C07129=5344,30396,-30623,463,-27004,-2829
C07130=5352,30386,-30635,462,-27000,-2833
C07131=5354,30373,-30650,461,-26996,-2833
C07132=5355,30360,-30666,461,-26991,-2834
C07133=5361,30350,-30679,461,-26987,-2836
C07134=5368,30340,-30691,460,-26983,-2839
C07135=5370,30327,-30707,459,-26978,-2840
C07136=5374,30315,-30721,459,-26974,-2841
C07137=5383,30306,-30731,458,-26971,-2845
C07138=5385,30293,-30747,457,-26966,-2846
C07139=5393,30284,-30758,456,-26963,-2849
C07140=5398,30273,-30772,456,-26958,-2851
C07141=5409,30265,-30781,454,-26956,-2855
C07142=5413,30254,-30795,454,-26951,-2857
C07143=5422,30245,-30806,452,-26948,-2860
C07144=5428,30234,-30818,451,-26944,-2863
C07145=5428,30229,-30825,451,-26942,-2863
C07146=5414,30227,-30827,454,-26941,-2857
C07147=5410,30239,-30813,454,-26946,-2856
C07148=5399,30246,-30804,456,-26949,-2851
C07149=5389,30255,-30793,457,-26952,-2848
C07150=5388,30268,-30778,457,-26957,-2847
C07151=5379,30277,-30767,458,-26960,-2843
C07152=5379,30277,-29367,458,-26960,-2843
C07153=5291,30621,-26350,469,-27087,-2808
C07154=5291,30621,-30350,469,-27087,-2808
C07155=5290,30633,-30335,469,-27092,-2807
C07156=5284,30643,-30323,470,-27096,-2805
C07157=5277,30652,-30312,471,-27099,-2802
C07158=5275,30665,-30298,471,-27104,-2802
C07159=5266,30673,-30288,472,-27107,-2798
C07160=5263,30684,-30275,473,-27111,-2797
C07161=5259,30695,-30261,473,-27115,-2795
C07162=5250,30703,-30251,474,-27118,-2792
C07163=5245,30713,-30239,475,-27121,-2790
C07164=5237,30722,-30228,476,-27125,-2787
C07165=5236,30734,-30214,476,-27129,-2786
C07166=5234,30746,-30199,476,-27134,-2785
C07167=5224,30754,-30190,478,-27136,-2781
C07168=5221,30765,-30176,478,-27141,-2780
C07169=5217,30776,-30163,479,-27145,-2778
C07170=5209,30785,-30153,480,-27148,-2775
C07171=5207,30797,-30138,480,-27152,-2775
C07172=5206,30809,-30123,480,-27157,-2774
C07173=5196,30817,-30114,482,-27160,-2770
C07174=5193,30828,-28700,482,-27164,-2769
C07175=-41004,59868,4099,4900,-34257,16705
C07176=-41004,59868,1099,4900,-34257,16705
C07177=-41004,64596,1380,5213,-31659,16463
C07178=-41004,59868,1099,4900,-34257,16705
C07179=-41004,59868,9099,4900,-34257,16705
C07180=5193,30828,-26100,482,-27164,-2769
C07181=5193,30828,-30100,482,-27164,-2769
C07182=5191,30840,-30085,482,-27168,-2768
C07183=5190,30853,-30070,482,-27173,-2768
C07184=5188,30865,-30055,482,-27178,-2767
C07185=5178,30872,-30047,484,-27180,-2763
C07186=5175,30884,-30032,484,-27185,-2762
C07187=5174,30896,-30018,484,-27189,-2761
C07188=5172,30908,-30003,484,-27194,-2761
C07189=5171,30921,-29988,484,-27198,-2760
C07190=5169,30933,-29973,485,-27203,-2759
C07191=5174,30934,-29971,484,-27203,-2761
C07192=5181,30925,-29983,483,-27200,-2764
C07193=5182,30913,-29997,483,-27195,-2764
C07194=5184,30900,-30012,483,-27191,-2765
C07195=5185,30888,-30027,483,-27186,-2766
C07196=5192,30879,-30038,482,-27183,-2768
C07197=5198,30869,-30050,481,-27179,-2771
C07198=5200,30857,-30065,481,-27175,-2771
C07199=5201,30845,-30080,481,-27170,-2772
C07200=5207,30835,-30092,480,-27166,-2774
C07201=5214,30826,-30103,479,-27163,-2777
C07202=5215,30813,-30118,479,-27159,-2778
C07203=5217,30801,-30132,478,-27154,-2779
C07204=5228,30794,-30141,477,-27151,-2783
C07205=5230,30782,-30156,477,-27147,-2783
C07206=5235,30772,-30168,476,-27143,-2785
C07207=5242,30763,-30179,475,-27140,-2788
C07208=5244,30751,-30193,475,-27135,-2789
C07209=5253,30742,-30203,474,-27132,-2792
C07210=5257,30732,-30217,473,-27128,-2794
C07211=5260,30720,-30230,473,-27124,-2795
C07212=5269,30712,-30240,471,-27121,-2799
C07213=5271,30700,-30254,471,-27117,-2800
C07214=5277,30691,-30266,470,-27113,-2802
C07215=5284,30681,-30278,470,-27110,-2805
C07216=5285,30669,-30292,469,-27105,-2805
C07217=5288,30657,-30306,469,-27101,-2807
C07218=5298,30650,-30315,468,-27098,-2810
C07219=5300,30638,-30330,468,-27094,-2811
C07220=5301,30625,-30345,467,-27089,-2812
C07221=5291,30621,-30350,469,-27087,-2808
C07222=5291,30621,-28950,469,-27087,-2808
C07223=5528,30636,-26331,434,-27095,-2900
C07224=5528,30636,-30331,434,-27095,-2900
C07225=5527,30651,-30313,434,-27101,-2899
C07226=5525,30666,-30295,434,-27106,-2898
C07227=5523,30681,-30277,435,-27112,-2897
C07228=5512,30691,-30265,436,-27115,-2893
C07229=5509,30705,-30248,436,-27121,-2892
C07230=5500,30716,-30234,438,-27124,-2888
C07231=5496,30729,-30218,438,-27129,-2887
C07232=5494,30744,-30200,438,-27135,-2886
C07233=5483,30754,-30189,440,-27138,-2881
C07234=5477,30766,-30173,441,-27143,-2879
C07235=5469,30778,-30160,442,-27147,-2876
C07236=5465,30792,-30143,442,-27152,-2875
C07237=5455,30802,-30130,444,-27156,-2871
C07238=5453,30817,-30112,444,-27162,-2870
C07239=5442,30826,-30101,445,-27165,-2865
C07240=5440,30841,-30083,446,-27171,-2865
C07241=5429,30851,-30071,447,-27174,-2860
C07242=5426,30865,-30054,447,-27180,-2859
C07243=5417,30876,-30041,449,-27184,-2856
C07244=5412,30889,-30025,449,-27188,-2853
C07245=5401,30899,-30013,451,-27192,-2849
C07246=5399,30914,-29995,451,-27198,-2849
C07247=5394,30927,-29979,452,-27202,-2846
C07248=5386,30938,-29966,453,-27206,-2843
C07249=5384,30953,-29948,453,-27212,-2842
C07250=5382,30968,-29930,453,-27218,-2842
C07251=5391,30980,-29915,452,-27222,-2845
C07252=5389,30995,-29897,452,-27228,-2844
C07253=5387,31010,-29879,452,-27233,-2843
C07254=5392,31014,-29874,452,-27235,-2845
C07255=5399,31002,-29888,451,-27230,-2848
C07256=5400,30987,-29906,450,-27225,-2849
C07257=5402,30972,-29924,450,-27219,-2849
C07258=5404,30957,-29942,450,-27214,-2850
C07259=5406,30942,-29960,450,-27208,-2851
C07260=5413,30930,-29975,449,-27204,-2854
C07261=5420,30918,-29990,448,-27199,-2856
C07262=5421,30903,-30007,448,-27194,-2857
C07263=5431,30893,-30020,447,-27190,-2861
C07264=5435,30879,-30037,446,-27185,-2862
C07265=5442,30867,-30051,445,-27181,-2865
C07266=5448,30855,-30066,444,-27176,-2868
C07267=5454,30842,-30082,444,-27171,-2870
C07268=5462,30831,-30095,443,-27167,-2873
C07269=5466,30817,-30112,442,-27162,-2875
C07270=5475,30806,-30125,441,-27158,-2878
C07271=5484,30795,-30138,439,-27154,-2882
C07272=5489,30782,-30154,439,-27149,-2884
C07273=5496,30770,-30169,438,-27145,-2887
C07274=5502,30758,-30183,437,-27140,-2889
C07275=5508,30745,-30199,436,-27135,-2891
C07276=5516,30734,-30213,435,-27131,-2894
C07277=5519,30720,-30230,435,-27126,-2896
C07278=5529,30709,-30242,433,-27122,-2900
C07279=5531,30695,-30260,433,-27117,-2901
C07280=5537,30682,-30276,433,-27112,-2903
C07281=5545,30670,-30289,431,-27108,-2906
C07282=5547,30656,-30307,431,-27102,-2907
C07283=5542,30642,-30324,432,-27097,-2905
C07284=5528,30636,-30331,434,-27095,-2900
C07285=5528,30636,-28931,434,-27095,-2900
C07286=5871,30873,-26043,382,-27186,-3031
C07287=5871,30873,-30043,382,-27186,-3031
C07288=5877,30878,-30036,381,-27188,-3034
C07289=5889,30880,-30034,380,-27189,-3038
C07290=5901,30882,-30031,378,-27190,-3043
C07291=5912,30883,-30029,376,-27190,-3047
C07292=5924,30885,-30027,375,-27191,-3052
C07293=5936,30887,-30025,373,-27192,-3056
C07294=5947,30888,-30023,371,-27193,-3061
C07295=5959,30890,-30021,369,-27193,-3065
C07296=5971,30892,-30019,368,-27194,-3070
C07297=5982,30894,-30017,366,-27195,-3074
C07298=5994,30895,-30015,364,-27195,-3079
C07299=6006,30897,-30012,363,-27196,-3083
C07300=6018,30899,-30010,361,-27197,-3088
C07301=6029,30900,-30008,359,-27198,-3093
C07302=6041,30902,-30006,357,-27198,-3097
C07303=6053,30904,-30004,356,-27199,-3102
C07304=6064,30906,-30002,354,-27200,-3106
C07305=6071,30914,-29991,353,-27203,-3109
C07306=6079,30923,-29980,352,-27207,-3112
C07307=6081,30933,-29968,351,-27210,-3112
C07308=6080,30944,-29955,351,-27214,-3112
C07309=6078,30955,-29942,352,-27218,-3111
C07310=6069,30961,-29934,353,-27221,-3108
C07311=6060,30968,-29926,354,-27223,-3104
C07312=6054,30976,-29916,355,-27226,-3102
C07313=6053,30987,-29903,355,-27230,-3101
C07314=6051,30998,-29890,355,-27234,-3101
C07315=6061,31001,-29886,354,-27235,-3105
C07316=6071,30994,-29894,352,-27233,-3108
C07317=6080,30988,-29902,351,-27231,-3112
C07318=6089,30981,-29910,350,-27228,-3116
C07319=6099,30975,-29917,348,-27226,-3119
C07320=6107,30968,-29925,347,-27224,-3122
C07321=6099,30960,-29936,348,-27220,-3119
C07322=6100,30949,-29949,349,-27216,-3120
C07323=6101,30938,-29962,348,-27212,-3120
C07324=6100,30928,-29974,349,-27209,-3120
C07325=6093,30919,-29985,350,-27205,-3117
C07326=6095,30908,-29998,349,-27201,-3118
C07327=6093,30900,-30008,350,-27198,-3117
C07328=6081,30898,-30011,352,-27197,-3113
C07329=6072,30893,-30017,353,-27195,-3109
C07330=6063,30886,-30025,354,-27193,-3106
C07331=6051,30884,-30027,356,-27192,-3101
C07332=6040,30883,-30030,358,-27191,-3097
C07333=6028,30881,-30032,359,-27190,-3092
C07334=6016,30879,-30034,361,-27190,-3088
C07335=6005,30878,-30036,363,-27189,-3083
C07336=5993,30876,-30038,365,-27188,-3079
C07337=5981,30874,-30040,366,-27188,-3074
C07338=5969,30873,-30042,368,-27187,-3069
C07339=5958,30871,-30044,370,-27186,-3065
C07340=5946,30869,-30046,371,-27185,-3060
C07341=5934,30867,-30049,373,-27185,-3056
C07342=5925,30874,-30041,374,-27187,-3052
C07343=5914,30874,-30041,376,-27187,-3048
C07344=5902,30872,-30043,378,-27186,-3043
C07345=5890,30871,-30045,380,-27185,-3039
C07346=5879,30869,-30047,381,-27185,-3034
C07347=5871,30873,-28643,382,-27186,-3031
C07348=-41004,59868,4099,4900,-34257,16705
C07349=-41004,59868,1099,4900,-34257,16705
C07350=-41004,64596,1380,5213,-31659,16463
C07351=-41004,59868,1099,4900,-34257,16705
C07352=-41004,59868,9099,4900,-34257,16705
C07353=5871,30873,-26043,382,-27186,-3031
C07354=5871,30873,-30043,382,-27186,-3031
C07355=5871,30873,-28643,382,-27186,-3031
C07356=5732,31221,-25621,401,-27315,-2976
C07357=5732,31221,-29621,401,-27315,-2976
C07358=5695,31216,-29627,406,-27313,-2962
C07359=5657,31210,-29634,412,-27310,-2947
C07360=5620,31205,-29641,417,-27308,-2933
C07361=5583,31200,-29648,422,-27306,-2918
C07362=5546,31194,-29654,428,-27303,-2904
C07363=5509,31189,-29661,433,-27301,-2890
C07364=5475,31193,-29656,438,-27303,-2876
C07365=5437,31188,-29662,444,-27300,-2862
C07366=5401,31187,-29664,449,-27300,-2848
C07367=5366,31187,-29664,454,-27299,-2834
C07368=5332,31193,-29657,459,-27301,-2821
C07369=5298,31196,-29653,464,-27302,-2808
C07370=5264,31201,-29647,469,-27304,-2795
C07371=5229,31206,-29642,474,-27305,-2781
C07372=5196,31211,-29635,479,-27307,-2768
C07373=5164,31225,-29619,483,-27312,-2756
C07374=5130,31230,-29614,488,-27313,-2743
C07375=5099,31244,-29596,493,-27318,-2731
C07376=5065,31249,-29591,498,-27320,-2717
C07377=5032,31258,-29580,502,-27323,-2705
C07378=5000,31268,-29568,507,-27326,-2692
C07379=4967,31278,-29556,512,-27330,-2679
C07380=4945,31289,-29543,515,-27334,-2671
C07381=4979,31284,-29548,510,-27332,-2684
C07382=5011,31272,-29562,505,-27328,-2696
C07383=5045,31265,-29571,500,-27326,-2709
C07384=5079,31260,-29577,496,-27324,-2723
C07385=5112,31253,-29585,491,-27322,-2736
C07386=5144,31241,-29600,486,-27318,-2748
C07387=5178,31236,-29605,481,-27316,-2761
C07388=5212,31232,-29610,476,-27315,-2774
C07389=5246,31227,-29616,471,-27313,-2788
C07390=5280,31223,-29621,466,-27312,-2801
C07391=5314,31218,-29627,461,-27310,-2814
C07392=5349,31213,-29632,457,-27309,-2827
C07393=5385,31216,-29629,451,-27310,-2842
C07394=5420,31214,-29631,446,-27310,-2855
C07395=5454,31210,-29636,441,-27309,-2868
C07396=5490,31211,-29635,436,-27309,-2882
C07397=5525,31210,-29635,431,-27309,-2896
C07398=5563,31216,-29628,425,-27312,-2910
C07399=5600,31221,-29621,420,-27314,-2925
C07400=5637,31227,-29615,414,-27316,-2939
C07401=5674,31232,-29608,409,-27319,-2954
C07402=5711,31237,-29601,404,-27321,-2968
C07403=5748,31243,-29594,398,-27323,-2982
C07404=5785,31248,-29588,393,-27326,-2997
C07405=5823,31254,-29581,387,-27328,-3011
C07406=5854,31268,-29564,382,-27334,-3023
C07407=5892,31273,-29557,377,-27336,-3038
C07408=5923,31287,-29539,372,-27341,-3050
C07409=5960,31293,-29532,367,-27344,-3064
C07410=5974,31288,-29538,365,-27342,-3070
C07411=5939,31279,-29550,370,-27338,-3056
C07412=5907,31266,-29566,375,-27333,-3044
C07413=5875,31252,-29583,380,-27328,-3031
C07414=5838,31246,-29590,385,-27325,-3017
C07415=5801,31240,-29597,390,-27323,-3003
C07416=5769,31227,-29614,395,-27317,-2990
C07417=5732,31221,-29621,401,-27315,-2976
C07418=5732,31221,-28221,401,-27315,-2976
C07419=4765,31119,-25749,542,-27269,-2602
C07420=4765,31119,-29749,542,-27269,-2602
C07421=4766,31110,-29761,542,-27265,-2602
C07422=4760,31102,-29770,543,-27262,-2600
C07423=4758,31094,-29780,543,-27259,-2599
C07424=4759,31085,-29791,543,-27256,-2599
C07425=4760,31075,-29802,543,-27252,-2600
C07426=4764,31068,-29811,543,-27250,-2602
C07427=4772,31062,-29818,542,-27248,-2605
C07428=4773,31053,-29829,542,-27244,-2605
C07429=4763,31052,-29831,543,-27244,-2601
C07430=4755,31057,-29824,544,-27246,-2598
C07431=4751,31065,-29815,545,-27248,-2596
C07432=4750,31074,-29804,545,-27252,-2596
C07433=4749,31083,-29793,545,-27255,-2595
C07434=4747,31093,-29782,545,-27259,-2595
C07435=4746,31102,-29770,545,-27262,-2595
C07436=4745,31111,-29759,545,-27266,-2594
C07437=4744,31120,-29748,545,-27269,-2594
C07438=4743,31129,-29737,545,-27272,-2593
C07439=4739,31137,-29728,546,-27275,-2592
C07440=4732,31143,-29721,547,-27277,-2589
C07441=4730,31152,-29710,547,-27281,-2588
C07442=4729,31161,-29699,547,-27284,-2588
C07443=4722,31167,-29692,548,-27286,-2585
C07444=4717,31174,-29683,549,-27289,-2583
C07445=4713,31182,-29674,549,-27292,-2581
C07446=4705,31187,-29667,550,-27294,-2578
C07447=4704,31196,-29656,550,-27297,-2578
C07448=4697,31202,-29649,551,-27299,-2575
C07449=4693,31210,-29640,552,-27302,-2573
C07450=4688,31217,-29631,553,-27305,-2571
C07451=4681,31223,-29624,554,-27307,-2568
C07452=4679,31232,-29614,554,-27310,-2568
C07453=4671,31237,-29607,555,-27312,-2565
C07454=4668,31245,-29597,555,-27315,-2563
C07455=4663,31252,-29589,556,-27317,-2561
C07456=4656,31258,-29582,557,-27320,-2559
C07457=4655,31267,-29570,557,-27323,-2558
C07458=4655,31274,-29562,557,-27326,-2558
C07459=4663,31269,-29568,556,-27324,-2561
C07460=4671,31263,-29575,555,-27322,-2564
C07461=4677,31257,-29583,554,-27319,-2567
C07462=4679,31249,-29593,554,-27316,-2568
C07463=4687,31243,-29600,553,-27314,-2571
C07464=4690,31235,-29610,552,-27311,-2572
C07465=4696,31228,-29617,551,-27309,-2574
C07466=4701,31222,-29626,551,-27306,-2576
C07467=4705,31214,-29635,550,-27303,-2578
C07468=4712,31208,-29642,549,-27301,-2581
C07469=4714,31199,-29653,549,-27298,-2582
C07470=4721,31193,-29660,548,-27296,-2584
C07471=4726,31186,-29668,547,-27293,-2586
C07472=4730,31178,-29678,547,-27291,-2588
C07473=4738,31173,-29684,546,-27289,-2591
C07474=4739,31164,-29695,546,-27285,-2591
C07475=4746,31158,-29702,545,-27283,-2594
C07476=4751,31151,-29711,544,-27280,-2596
C07477=4752,31141,-29722,544,-27277,-2597
C07478=4753,31132,-29734,544,-27274,-2597
C07479=4757,31125,-29743,543,-27271,-2599
C07480=4765,31119,-29749,542,-27269,-2602
C07481=4765,31119,-28349,542,-27269,-2602
C07482=3339,30279,-26773,757,-26945,-2054
C07483=3339,30279,-30773,757,-26945,-2054
C07484=3349,30265,-30790,756,-26939,-2058
C07485=3361,30252,-30806,754,-26935,-2062
C07486=3371,30239,-30822,753,-26930,-2067
C07487=3380,30224,-30840,752,-26924,-2070
C07488=3386,30208,-30860,751,-26918,-2072
C07489=3397,30194,-30876,750,-26914,-2077
C07490=3405,30180,-30894,749,-26908,-2080
C07491=3413,30165,-30911,748,-26903,-2083
C07492=3416,30152,-30927,747,-26898,-2084
C07493=3411,30135,-30947,748,-26892,-2082
C07494=3405,30119,-30968,749,-26885,-2080
C07495=3396,30103,-30987,751,-26879,-2077
C07496=3387,30087,-31006,752,-26873,-2074
C07497=3389,30068,-31028,752,-26867,-2075
C07498=3391,30050,-31051,752,-26860,-2075
C07499=3393,30031,-31073,752,-26853,-2076
C07500=3394,30013,-31095,752,-26846,-2077
C07501=3402,29998,-31114,751,-26841,-2080
C07502=3408,29982,-31133,750,-26835,-2082
C07503=3410,29963,-31155,750,-26828,-2083
C07504=3411,29945,-31178,750,-26821,-2084
C07505=3413,29926,-31200,750,-26814,-2085
C07506=3415,29908,-31222,750,-26807,-2086
C07507=3424,29894,-31239,749,-26802,-2089
C07508=3429,29877,-31260,748,-26796,-2091
C07509=3430,29858,-31282,748,-26789,-2092
C07510=3432,29840,-31304,748,-26782,-2093
C07511=3430,29822,-31326,748,-26776,-2092
C07512=3414,29813,-31336,751,-26772,-2086
C07513=3412,29832,-31314,751,-26779,-2085
C07514=3410,29850,-31292,751,-26786,-2084
C07515=3408,29869,-31270,751,-26793,-2083
C07516=3407,29887,-31248,751,-26800,-2083
C07517=3405,29905,-31225,751,-26806,-2082
C07518=3398,29921,-31206,752,-26812,-2079
C07519=3391,29937,-31187,753,-26818,-2076
C07520=3390,29955,-31165,753,-26825,-2076
C07521=3388,29974,-31143,753,-26832,-2075
C07522=3385,29992,-31121,753,-26838,-2074
C07523=3374,30005,-29705,755,-26843,-2069
C07524=-41004,59868,4099,4900,-34257,16705
C07525=-41004,59868,1099,4900,-34257,16705
C07526=-41004,64596,1380,5213,-31659,16463
C07527=-41004,59868,1099,4900,-34257,16705
C07528=-41004,59868,9099,4900,-34257,16705
C07529=3374,30005,-27105,755,-26843,-2069
C07530=3374,30005,-31105,755,-26843,-2069
C07531=3373,30023,-31083,755,-26850,-2069
C07532=3371,30042,-31060,755,-26857,-2068
C07533=3369,30060,-31038,755,-26864,-2067
C07534=3367,30079,-31016,755,-26870,-2066
C07535=3366,30097,-30994,755,-26877,-2065
C07536=3374,30113,-30974,754,-26883,-2068
C07537=3387,30128,-30956,752,-26889,-2073
C07538=3392,30145,-30936,751,-26895,-2075
C07539=3397,30159,-30919,750,-26900,-2077
C07540=3389,30174,-30901,751,-26906,-2074
C07541=3378,30187,-30885,753,-26911,-2069
C07542=3372,30203,-30865,753,-26917,-2067
C07543=3364,30218,-30847,754,-26922,-2064
C07544=3355,30233,-30830,755,-26927,-2060
C07545=3341,30244,-30816,757,-26932,-2055
C07546=3331,30258,-30799,759,-26937,-2051
C07547=3327,30276,-30778,759,-26943,-2049
C07548=3316,30289,-30762,761,-26948,-2045
C07549=3324,30290,-30760,759,-26948,-2048
C07550=3339,30279,-30773,757,-26945,-2054
C07551=3339,30279,-29373,757,-26945,-2054
C07552=3255,30276,-26778,770,-26943,-2021
C07553=3255,30276,-30778,770,-26943,-2021
C07554=3257,30254,-30805,770,-26934,-2022
C07555=3266,30235,-30827,768,-26928,-2026
C07556=3271,30215,-30852,768,-26920,-2028
C07557=3282,30197,-30873,766,-26914,-2032
C07558=3283,30177,-30897,766,-26906,-2033
C07559=3263,30185,-30888,769,-26909,-2025
C07560=3246,30184,-30889,772,-26908,-2018
C07561=3245,30162,-30916,772,-26900,-2018
C07562=3247,30140,-30942,772,-26892,-2019
C07563=3249,30118,-30969,772,-26884,-2020
C07564=3259,30099,-30991,771,-26877,-2024
C07565=3273,30084,-31010,769,-26872,-2030
C07566=3275,30062,-31037,769,-26863,-2031
C07567=3267,30042,-31061,770,-26856,-2028
C07568=3260,30022,-31085,771,-26848,-2025
C07569=3261,30000,-31112,772,-26840,-2025
C07570=3263,29978,-31138,771,-26832,-2026
C07571=3265,29956,-31165,771,-26824,-2027
C07572=3276,29938,-31186,770,-26818,-2032
C07573=3279,29917,-31212,770,-26810,-2033
C07574=3281,29894,-31239,770,-26801,-2034
C07575=3273,29875,-31263,771,-26794,-2031
C07576=3275,29852,-31290,771,-26786,-2032
C07577=3268,29832,-31314,772,-26778,-2029
C07578=3260,29812,-31339,774,-26771,-2026
C07579=3259,29791,-31365,774,-26763,-2026
C07580=3240,29779,-31379,777,-26758,-2019
C07581=3241,29800,-31353,776,-26766,-2019
C07582=3249,29820,-31329,775,-26774,-2022
C07583=3255,29841,-31304,774,-26781,-2024
C07584=3253,29863,-31278,774,-26789,-2023
C07585=3251,29885,-31251,774,-26798,-2022
C07586=3249,29907,-31224,774,-26806,-2021
C07587=3246,29929,-31197,774,-26814,-2020
C07588=3244,29952,-31170,774,-26822,-2019
C07589=3242,29974,-31143,774,-26831,-2018
C07590=3240,29996,-31116,775,-26839,-2017
C07591=3246,30016,-31092,773,-26846,-2020
C07592=3247,30038,-31066,773,-26854,-2020
C07593=3255,30058,-31042,772,-26862,-2023
C07594=3251,30079,-31016,772,-26870,-2021
C07595=3241,30097,-30995,773,-26876,-2017
C07596=3235,30117,-30970,774,-26883,-2015
C07597=3227,30136,-30947,775,-26890,-2011
C07598=3235,30156,-30923,774,-26898,-2015
C07599=3233,30178,-30897,774,-26906,-2014
C07600=3240,30198,-30872,773,-26914,-2016
C07601=3240,30220,-30846,772,-26922,-2016
C07602=3237,30242,-30819,773,-26930,-2015
C07603=3235,30264,-30792,773,-26938,-2014
C07604=3232,30286,-30766,773,-26946,-2012
C07605=3220,30303,-30746,774,-26952,-2008
C07606=3202,30316,-30730,777,-26957,-2000
C07607=3183,30329,-30714,780,-26962,-1993
C07608=3182,30344,-30696,780,-26967,-1992
C07609=3202,30338,-30704,777,-26965,-2000
C07610=3222,30328,-30715,774,-26962,-2008
C07611=3240,30315,-30731,771,-26957,-2015
C07612=3252,30298,-30751,770,-26951,-2020
C07613=3255,30276,-30778,770,-26943,-2021
C07614=3255,30276,-29378,770,-26943,-2021
C07615=2834,30120,-26969,833,-26881,-1859
C07616=2834,30120,-30969,833,-26881,-1859
C07617=2846,30102,-30990,831,-26875,-1864
C07618=2858,30084,-31011,830,-26868,-1869
C07619=2860,30061,-31039,829,-26860,-1870
C07620=2870,30043,-31062,828,-26853,-1874
C07621=2876,30021,-31088,828,-26845,-1876
C07622=2886,30003,-31110,826,-26838,-1880
C07623=2888,29980,-31138,826,-26830,-1881
C07624=2891,29957,-31165,826,-26821,-1882
C07625=2889,29935,-31192,827,-26813,-1882
C07626=2869,29922,-31208,830,-26808,-1874
C07627=2864,29901,-31234,831,-26800,-1873
C07628=2866,29878,-31261,831,-26792,-1874
C07629=2858,29857,-31286,832,-26784,-1870
C07630=2860,29834,-31314,832,-26776,-1871
C07631=2872,29816,-31336,830,-26769,-1876
C07632=2881,29797,-31359,829,-26762,-1880
C07633=2875,29783,-31375,830,-26757,-1878
C07634=2863,29801,-31354,832,-26763,-1873
C07635=2851,29819,-31333,833,-26770,-1868
C07636=2849,29842,-31305,833,-26778,-1867
C07637=2847,29865,-31277,834,-26787,-1866
C07638=2848,29887,-31250,833,-26795,-1866
C07639=2856,29908,-31225,832,-26803,-1870
C07640=2872,29927,-31202,829,-26810,-1876
C07641=2874,29949,-31175,829,-26818,-1876
C07642=2879,29970,-31149,828,-26826,-1878
C07643=2877,29993,-31121,828,-26835,-1877
C07644=2865,30011,-31100,829,-26841,-1872
C07645=2860,30033,-31074,830,-26849,-1870
C07646=2851,30052,-31051,831,-26856,-1866
C07647=2843,30072,-31027,832,-26864,-1863
C07648=2830,30089,-31006,834,-26870,-1858
C07649=2818,30107,-30985,835,-26876,-1853
C07650=2799,30120,-30968,838,-26881,-1846
C07651=2787,30138,-30947,839,-26888,-1841
C07652=2769,30152,-30930,842,-26893,-1834
C07653=2756,30169,-30909,844,-26899,-1829
C07654=2744,30187,-30888,845,-26905,-1824
C07655=2734,30205,-30866,846,-26912,-1820
C07656=2722,30223,-30844,848,-26919,-1815
C07657=2720,30246,-30816,848,-26927,-1814
C07658=2718,30269,-30789,848,-26936,-1813
C07659=2716,30292,-30761,848,-26944,-1812
C07660=2714,30315,-30733,848,-26953,-1811
C07661=2712,30338,-30705,848,-26961,-1810
C07662=2700,30356,-30684,850,-26968,-1806
C07663=2706,30364,-30674,849,-26971,-1808
C07664=2721,30348,-30693,847,-26965,-1814
C07665=2723,30325,-30721,847,-26956,-1815
C07666=2725,30302,-30749,847,-26948,-1816
C07667=2727,30279,-30777,847,-26939,-1817
C07668=2729,30256,-30805,847,-26931,-1818
C07669=2741,30238,-30826,845,-26924,-1822
C07670=2743,30215,-30854,845,-26916,-1823
C07671=2755,30197,-30875,843,-26909,-1828
C07672=2767,30180,-30897,842,-26903,-1833
C07673=2785,30166,-30914,839,-26898,-1840
C07674=2798,30148,-30935,838,-26891,-1845
C07675=2817,30134,-30951,835,-26887,-1853
C07676=2834,30120,-30969,833,-26881,-1859
C07677=2834,30120,-29569,833,-26881,-1859
C07678=2940,29896,-27239,820,-26799,-1902
C07679=2940,29896,-31239,820,-26799,-1902
C07680=2954,29868,-31272,818,-26789,-1907
C07681=2964,29839,-31308,817,-26778,-1911
C07682=2975,29809,-31343,815,-26767,-1916
C07683=2980,29777,-31383,815,-26755,-1918
C07684=2983,29743,-31423,815,-26743,-1920
C07685=2986,29710,-31464,815,-26731,-1921
C07686=2989,29676,-31504,815,-26718,-1922
C07687=2981,29645,-31542,816,-26707,-1920
C07688=2972,29614,-31579,818,-26695,-1916
C07689=2956,29585,-31614,820,-26684,-1910
C07690=2940,29556,-31650,823,-26673,-1904
C07691=2931,29525,-31687,825,-26662,-1901
C07692=2922,29494,-31724,826,-26650,-1898
C07693=2925,29461,-31765,826,-26638,-1899
C07694=2917,29430,-31802,828,-26626,-1896
C07695=2920,29396,-31843,828,-26614,-1898
C07696=2923,29363,-31884,828,-26602,-1899
C07697=2936,29335,-31917,826,-26591,-1904
C07698=2949,29307,-31951,824,-26581,-1910
C07699=2962,29278,-30585,823,-26571,-1915
C07700=-41004,59868,4099,4900,-34257,16705
C07701=-41004,59868,1099,4900,-34257,16705
C07702=-41004,64596,1380,5213,-31659,16463
C07703=-41004,59868,1099,4900,-34257,16705
C07704=-41004,59868,9099,4900,-34257,16705
C07705=2962,29278,-27985,823,-26571,-1915
C07706=2962,29278,-31985,823,-26571,-1915
C07707=2975,29250,-32019,821,-26560,-1920
C07708=2988,29222,-32053,819,-26550,-1925
C07709=2991,29189,-32094,819,-26538,-1927
C07710=3004,29161,-32128,818,-26527,-1932
C07711=3007,29127,-32168,818,-26515,-1933
C07712=3010,29093,-32209,818,-26503,-1935
C07713=3013,29060,-32249,817,-26490,-1936
C07714=3016,29026,-32290,817,-26478,-1938
C07715=3019,28993,-32330,817,-26465,-1939
C07716=3000,28970,-32358,820,-26457,-1932
C07717=3008,29001,-32321,819,-26468,-1935
C07718=3005,29034,-32280,819,-26481,-1933
C07719=3002,29068,-32240,819,-26493,-1932
C07720=2999,29101,-32199,819,-26505,-1930
C07721=2996,29135,-32159,819,-26518,-1929
C07722=2987,29165,-32122,820,-26529,-1925
C07723=2980,29197,-32084,821,-26541,-1922
C07724=2967,29225,-32050,823,-26551,-1917
C07725=2954,29253,-32016,824,-26561,-1912
C07726=2941,29281,-31982,826,-26571,-1907
C07727=2928,29309,-31948,827,-26582,-1901
C07728=2905,29332,-31921,831,-26590,-1892
C07729=2902,29365,-31881,831,-26602,-1891
C07730=2899,29399,-31840,831,-26615,-1890
C07731=2896,29432,-31799,831,-26627,-1888
C07732=2904,29464,-31762,829,-26639,-1891
C07733=2906,29496,-31723,829,-26651,-1891
C07734=2914,29527,-31685,827,-26662,-1895
C07735=2927,29557,-31649,825,-26674,-1899
C07736=2939,29587,-31613,823,-26685,-1904
C07737=2955,29616,-31577,820,-26696,-1910
C07738=2960,29648,-31539,819,-26707,-1911
C07739=2968,29679,-31501,818,-26719,-1914
C07740=2965,29712,-31461,818,-26731,-1913
C07741=2962,29746,-31420,818,-26744,-1911
C07742=2969,29777,-31383,816,-26755,-1914
C07743=2956,29805,-31349,818,-26766,-1909
C07744=2943,29833,-31315,820,-26776,-1904
C07745=2940,29867,-31274,820,-26788,-1902
C07746=2940,29896,-31239,820,-26799,-1902
C07747=2940,29896,-29839,820,-26799,-1902
C07748=2704,29594,-27605,857,-26685,-1813
C07749=2704,29594,-31605,857,-26685,-1813
C07750=2715,29588,-31612,856,-26684,-1817
C07751=2721,29575,-31628,855,-26679,-1820
C07752=2734,29565,-31639,853,-26675,-1825
C07753=2739,29551,-31656,853,-26670,-1827
C07754=2747,29539,-31671,852,-26666,-1830
C07755=2752,29525,-31688,851,-26660,-1832
C07756=2759,29512,-31704,850,-26656,-1835
C07757=2765,29498,-31720,849,-26651,-1837
C07758=2766,29482,-31739,849,-26645,-1838
C07759=2767,29467,-31759,849,-26639,-1838
C07760=2769,29451,-31778,849,-26633,-1839
C07761=2770,29435,-31797,849,-26627,-1840
C07762=2772,29419,-31816,849,-26621,-1840
C07763=2764,29405,-31833,851,-26616,-1837
C07764=2764,29389,-31852,851,-26610,-1837
C07765=2774,29378,-31866,849,-26606,-1841
C07766=2776,29363,-31884,849,-26601,-1843
C07767=2778,29347,-31903,849,-26595,-1843
C07768=2785,29334,-31918,848,-26590,-1846
C07769=2791,29321,-31935,848,-26585,-1848
C07770=2792,29305,-31954,848,-26579,-1849
C07771=2803,29294,-31967,846,-26575,-1853
C07772=2805,29278,-31986,846,-26570,-1854
C07773=2806,29262,-32005,846,-26564,-1855
C07774=2816,29251,-32019,845,-26559,-1858
C07775=2819,29236,-32037,844,-26554,-1860
C07776=2821,29221,-32056,844,-26548,-1861
C07777=2832,29210,-32069,843,-26544,-1865
C07778=2841,29198,-32083,842,-26540,-1869
C07779=2841,29186,-32098,842,-26536,-1869
C07780=2824,29183,-32101,844,-26534,-1862
C07781=2817,29197,-32085,845,-26539,-1860
C07782=2811,29210,-32069,846,-26544,-1857
C07783=2810,29226,-32050,846,-26550,-1856
C07784=2799,29236,-32037,847,-26554,-1852
C07785=2797,29252,-32018,847,-26560,-1851
C07786=2793,29267,-32000,848,-26565,-1850
C07787=2784,29278,-31986,849,-26569,-1846
C07788=2783,29294,-31967,849,-26575,-1845
C07789=2775,29307,-31952,850,-26580,-1842
C07790=2770,29321,-31935,851,-26585,-1840
C07791=2768,29337,-31916,851,-26591,-1840
C07792=2757,29347,-31903,852,-26595,-1835
C07793=2756,29363,-31884,852,-26601,-1834
C07794=2754,29379,-31865,852,-26606,-1834
C07795=2753,29395,-31845,852,-26612,-1833
C07796=2751,29411,-31826,852,-26618,-1832
C07797=2750,29427,-31807,852,-26624,-1832
C07798=2751,29442,-31788,852,-26630,-1832
C07799=2758,29456,-31771,851,-26635,-1835
C07800=2755,29471,-31753,851,-26641,-1833
C07801=2745,29482,-31740,853,-26645,-1830
C07802=2744,29498,-31720,853,-26651,-1829
C07803=2736,29511,-31705,854,-26655,-1826
C07804=2731,29525,-31688,854,-26660,-1824
C07805=2730,29541,-31669,854,-26666,-1823
C07806=2718,29551,-31657,856,-26670,-1819
C07807=2717,29567,-31637,856,-26676,-1818
C07808=2705,29578,-31625,857,-26680,-1813
C07809=2704,29594,-31605,857,-26685,-1813
C07810=2704,29594,-30205,857,-26685,-1813
C07811=2496,29451,-27779,889,-26631,-1734
C07812=2496,29451,-31779,889,-26631,-1734
C07813=2462,29437,-31796,895,-26626,-1720
C07814=2422,29431,-31803,901,-26623,-1705
C07815=2383,29425,-31810,906,-26621,-1690
C07816=2344,29420,-31817,912,-26618,-1675
C07817=2304,29414,-31824,918,-26616,-1659
C07818=2265,29408,-31831,924,-26614,-1644
C07819=2225,29403,-31838,930,-26611,-1629
C07820=2191,29388,-31856,935,-26606,-1616
C07821=2152,29383,-31863,941,-26603,-1601
C07822=2112,29377,-31870,947,-26601,-1586
C07823=2077,29363,-31886,952,-26596,-1572
C07824=2039,29357,-31895,958,-26593,-1557
C07825=1999,29351,-31902,964,-26590,-1542
C07826=1960,29345,-31909,969,-26588,-1527
C07827=1920,29340,-31916,975,-26586,-1512
C07828=1881,29334,-31923,981,-26583,-1496
C07829=1842,29328,-31930,987,-26581,-1481
C07830=1802,29323,-31937,993,-26578,-1466
C07831=1763,29317,-31944,999,-26576,-1451
C07832=1723,29311,-31951,1005,-26574,-1436
C07833=1684,29305,-31958,1010,-26571,-1420
C07834=1648,29310,-31953,1016,-26572,-1407
C07835=1609,29304,-31960,1021,-26570,-1391
C07836=1570,29298,-31967,1027,-26568,-1376
C07837=1530,29293,-31974,1033,-26565,-1361
C07838=1491,29287,-31981,1039,-26563,-1346
C07839=1451,29281,-31988,1045,-26560,-1331
C07840=1416,29286,-31983,1050,-26562,-1317
C07841=1381,29271,-32001,1055,-26556,-1304
C07842=1363,29288,-31981,1058,-26562,-1296
C07843=1403,29293,-31974,1052,-26565,-1312
C07844=1442,29299,-31967,1046,-26567,-1327
C07845=1481,29305,-31960,1040,-26569,-1342
C07846=1521,29311,-31953,1034,-26572,-1357
C07847=1560,29315,-31947,1029,-26574,-1372
C07848=1596,29312,-31951,1023,-26573,-1386
C07849=1635,29318,-31944,1017,-26575,-1401
C07850=1675,29323,-31937,1012,-26578,-1417
C07851=1714,29329,-31930,1006,-26580,-1432
C07852=1753,29335,-31922,1000,-26582,-1447
C07853=1793,29340,-31915,994,-26585,-1462
C07854=1829,29336,-31921,989,-26583,-1476
C07855=1868,29342,-31914,983,-26586,-1491
C07856=1907,29347,-31907,977,-26588,-1506
C07857=1942,29362,-31889,972,-26594,-1520
C07858=1981,29367,-31882,966,-26596,-1535
C07859=2021,29373,-31875,960,-26599,-1550
C07860=2060,29379,-31868,954,-26601,-1565
C07861=2094,29393,-31850,949,-26607,-1578
C07862=2134,29399,-31843,943,-26609,-1594
C07863=2173,29405,-31836,937,-26612,-1609
C07864=2212,29410,-31829,932,-26614,-1624
C07865=2247,29425,-31811,926,-26620,-1637
C07866=2286,29431,-31804,921,-26622,-1652
C07867=2325,29436,-31797,915,-26624,-1668
C07868=2365,29442,-31790,909,-26627,-1683
C07869=2404,29448,-31783,903,-26629,-1698
C07870=2444,29453,-31776,897,-26632,-1713
C07871=2483,29459,-31769,891,-26634,-1728
C07872=2496,29451,-30379,889,-26631,-1734
C07873=-41004,59868,4099,4900,-34257,16705
C07874=-41004,59868,1099,4900,-34257,16705
C07875=-41004,64596,1380,5213,-31659,16463
C07876=-41004,59868,1099,4900,-34257,16705
C07877=-41004,59868,9099,4900,-34257,16705
C07878=2496,29451,-27779,889,-26631,-1734
C07879=2496,29451,-31779,889,-26631,-1734
C07880=2496,29451,-30379,889,-26631,-1734
C07881=2369,29567,-27639,907,-26673,-1683
C07882=2369,29567,-31639,907,-26673,-1683
C07883=2274,29553,-31656,921,-26667,-1647
C07884=2184,29531,-31684,934,-26658,-1612
C07885=2094,29508,-31712,948,-26649,-1577
C07886=1999,29494,-31729,962,-26643,-1541
C07887=1909,29472,-31756,975,-26634,-1506
C07888=1813,29458,-31773,990,-26628,-1469
C07889=1721,29439,-31796,1003,-26621,-1434
C07890=1628,29422,-31818,1017,-26614,-1398
C07891=1533,29408,-31835,1031,-26608,-1361
C07892=1438,29394,-31852,1045,-26602,-1324
C07893=1343,29380,-31869,1060,-26596,-1288
C07894=1247,29367,-31886,1074,-26590,-1251
C07895=1156,29363,-31891,1087,-26588,-1216
C07896=1061,29349,-31908,1101,-26582,-1179
C07897=1018,29275,-31998,1108,-26555,-1163
C07898=937,29236,-32045,1121,-26540,-1132
C07899=847,29213,-32073,1134,-26531,-1097
C07900=799,29144,-32157,1142,-26505,-1079
C07901=824,29067,-32250,1140,-26477,-1090
C07902=839,28985,-32349,1139,-26446,-1096
C07903=855,28903,-32447,1137,-26416,-1103
C07904=859,28823,-32543,1138,-26387,-1106
C07905=822,28751,-32631,1144,-26360,-1092
C07906=785,28673,-32725,1151,-26331,-1078
C07907=768,28591,-32824,1154,-26301,-1073
C07908=709,28534,-32893,1164,-26280,-1050
C07909=729,28592,-32823,1160,-26301,-1058
C07910=765,28651,-32751,1154,-26323,-1071
C07911=780,28734,-32651,1151,-26354,-1076
C07912=840,28801,-32570,1141,-26379,-1098
C07913=845,28886,-32467,1139,-26410,-1100
C07914=820,28963,-32375,1142,-26438,-1089
C07915=804,29045,-32276,1143,-26468,-1082
C07916=789,29127,-32177,1144,-26498,-1076
C07917=807,29209,-32078,1140,-26529,-1082
C07918=889,29248,-32031,1128,-26544,-1113
C07919=982,29265,-32010,1114,-26551,-1149
C07920=1031,29340,-31920,1106,-26579,-1167
C07921=1041,29423,-31818,1103,-26610,-1171
C07922=982,29462,-31772,1111,-26623,-1147
C07923=906,29413,-31832,1123,-26605,-1119
C07924=953,29465,-31769,1116,-26624,-1136
C07925=1037,29498,-31728,1103,-26637,-1168
C07926=1052,29424,-31818,1102,-26610,-1175
C07927=1085,29362,-31892,1098,-26587,-1188
C07928=1180,29376,-31875,1083,-26593,-1225
C07929=1276,29390,-31858,1069,-26599,-1262
C07930=1371,29403,-31841,1055,-26605,-1298
C07931=1466,29417,-31824,1041,-26611,-1335
C07932=1561,29431,-31807,1027,-26616,-1372
C07933=1656,29445,-31790,1013,-26622,-1408
C07934=1751,29458,-31773,999,-26628,-1445
C07935=1841,29481,-31745,985,-26637,-1480
C07936=1937,29495,-31728,971,-26643,-1517
C07937=2027,29517,-31700,958,-26652,-1551
C07938=2122,29531,-31683,943,-26658,-1588
C07939=2212,29554,-31656,930,-26667,-1623
C07940=2307,29567,-31639,916,-26673,-1659
C07941=2397,29590,-31611,902,-26682,-1694
C07942=2369,29567,-31639,907,-26673,-1683
C07943=2369,29567,-30239,907,-26673,-1683
C07944=2358,29623,-27572,908,-26693,-1679
C07945=2358,29623,-31572,908,-26693,-1679
C07946=2344,29630,-31563,910,-26696,-1673
C07947=2327,29628,-31566,912,-26695,-1667
C07948=2310,29625,-31569,915,-26694,-1660
C07949=2293,29623,-31572,917,-26693,-1653
C07950=2276,29620,-31575,920,-26692,-1647
C07951=2259,29618,-31578,922,-26691,-1640
C07952=2241,29615,-31581,925,-26690,-1634
C07953=2224,29613,-31584,928,-26689,-1627
C07954=2207,29610,-31587,930,-26688,-1620
C07955=2190,29608,-31590,933,-26687,-1614
C07956=2173,29605,-31593,935,-26686,-1607
C07957=2156,29603,-31597,938,-26685,-1601
C07958=2142,29609,-31589,940,-26687,-1595
C07959=2125,29608,-31591,942,-26686,-1589
C07960=2108,29606,-31594,945,-26685,-1582
C07961=2091,29603,-31597,947,-26684,-1575
C07962=2074,29601,-31600,950,-26683,-1569
C07963=2056,29598,-31603,952,-26682,-1562
C07964=2039,29596,-31606,955,-26681,-1556
C07965=2022,29593,-31609,957,-26680,-1549
C07966=2005,29591,-31612,960,-26679,-1542
C07967=1988,29588,-31615,962,-26678,-1536
C07968=1971,29586,-31618,965,-26677,-1529
C07969=1954,29583,-31621,968,-26676,-1523
C07970=1937,29581,-31624,970,-26675,-1516
C07971=1919,29578,-31627,973,-26674,-1509
C07972=1902,29576,-31630,975,-26673,-1503
C07973=1885,29573,-31633,978,-26672,-1496
C07974=1887,29583,-31622,977,-26675,-1497
C07975=1904,29586,-31619,975,-26676,-1503
C07976=1921,29588,-31615,972,-26677,-1510
C07977=1938,29591,-31612,970,-26678,-1517
C07978=1956,29593,-31609,967,-26679,-1523
C07979=1973,29596,-31606,965,-26680,-1530
C07980=1990,29598,-31603,962,-26682,-1536
C07981=2003,29607,-31592,960,-26685,-1541
C07982=2019,29612,-31586,958,-26687,-1548
C07983=2036,29614,-31583,955,-26688,-1554
C07984=2053,29617,-31580,953,-26689,-1561
C07985=2067,29610,-31589,951,-26686,-1566
C07986=2084,29612,-31586,948,-26687,-1573
C07987=2101,29614,-31583,946,-26688,-1579
C07988=2118,29617,-31580,943,-26689,-1586
C07989=2135,29619,-31577,940,-26690,-1593
C07990=2152,29620,-31576,938,-26691,-1599
C07991=2166,29614,-31583,936,-26689,-1604
C07992=2183,29616,-31580,933,-26690,-1611
C07993=2200,29619,-31577,931,-26691,-1618
C07994=2218,29621,-31574,928,-26692,-1624
C07995=2235,29624,-31571,926,-26693,-1631
C07996=2252,29626,-31568,923,-26694,-1638
C07997=2269,29629,-31565,921,-26695,-1644
C07998=2286,29631,-31562,918,-26696,-1651
C07999=2303,29634,-31559,916,-26697,-1657
C08000=2320,29636,-31556,913,-26698,-1664
C08001=2337,29639,-31552,911,-26699,-1671
C08002=2355,29641,-31549,908,-26700,-1677
C08003=2368,29633,-31559,906,-26697,-1682
C08004=2375,29625,-31569,905,-26695,-1685
C08005=2358,29623,-31572,908,-26693,-1679
C08006=2358,29623,-30172,908,-26693,-1679
C08007=2763,29161,-28128,853,-26526,-1839
C08008=2763,29161,-32128,853,-26526,-1839
C08009=2771,29159,-32131,852,-26525,-1842
C08010=2776,29146,-32146,852,-26520,-1844
C08011=2786,29136,-32158,850,-26517,-1848
C08012=2793,29125,-32171,849,-26513,-1851
C08013=2798,29113,-32186,849,-26508,-1853
C08014=2800,29099,-32203,849,-26503,-1853
C08015=2808,29088,-32216,848,-26499,-1857
C08016=2804,29078,-32229,848,-26495,-1855
C08017=2803,29064,-32245,849,-26490,-1855
C08018=2804,29050,-32263,849,-26485,-1855
C08019=2805,29035,-32280,848,-26480,-1856
C08020=2806,29021,-32297,848,-26474,-1857
C08021=2798,29009,-32312,850,-26470,-1854
C08022=2796,28995,-32328,850,-26465,-1853
C08023=2789,28983,-32343,851,-26460,-1850
C08024=2790,28969,-32361,851,-26455,-1851
C08025=2781,28957,-32375,853,-26450,-1847
C08026=2778,28943,-32391,854,-26445,-1846
C08027=2772,28931,-32407,854,-26441,-1844
C08028=2774,28916,-32424,854,-26435,-1845
C08029=2775,28902,-32441,854,-26430,-1845
C08030=2776,28888,-32458,854,-26425,-1846
C08031=2777,28873,-32476,854,-26419,-1846
C08032=2778,28859,-32493,854,-26414,-1847
C08033=2780,28845,-32510,854,-26409,-1848
C08034=2783,28831,-32526,854,-26404,-1849
C08035=2792,28822,-32538,853,-26400,-1853
C08036=2794,28807,-32556,853,-26395,-1853
C08037=2795,28793,-32573,853,-26390,-1854
C08038=2802,28782,-32586,852,-26386,-1857
C08039=2796,28778,-32591,853,-26384,-1854
C08040=2791,28790,-32576,853,-26389,-1852
C08041=2784,28801,-32563,854,-26393,-1849
C08042=2781,28815,-32547,854,-26398,-1848
C08043=2771,28824,-32535,856,-26401,-1844
C08044=2770,28838,-32518,856,-26406,-1844
C08045=2769,28853,-32501,856,-26412,-1843
C08046=2767,28867,-32483,856,-26417,-1843
C08047=2766,28881,-32466,856,-26422,-1842
C08048=2765,28896,-31049,856,-26428,-1841
C08049=-41004,59868,4099,4900,-34257,16705
C08050=-41004,59868,1099,4900,-34257,16705
C08051=-41004,64596,1380,5213,-31659,16463
C08052=-41004,59868,1099,4900,-34257,16705
C08053=-41004,59868,9099,4900,-34257,16705
C08054=2765,28896,-28449,856,-26428,-1841
C08055=2765,28896,-32449,856,-26428,-1841
C08056=2764,28910,-32432,856,-26433,-1841
C08057=2762,28924,-32414,856,-26438,-1840
C08058=2761,28939,-32397,856,-26443,-1840
C08059=2766,28951,-32382,855,-26448,-1842
C08060=2769,28965,-32365,855,-26453,-1843
C08061=2772,28978,-32349,854,-26458,-1843
C08062=2778,28991,-32334,853,-26463,-1846
C08063=2777,29005,-32317,853,-26468,-1845
C08064=2786,29017,-32302,852,-26473,-1849
C08065=2785,29031,-32285,852,-26478,-1848
C08066=2785,29045,-32268,851,-26483,-1848
C08067=2793,29058,-32253,850,-26488,-1851
C08068=2791,29072,-32236,850,-26493,-1850
C08069=2790,29086,-32218,850,-26498,-1850
C08070=2789,29100,-32201,850,-26504,-1849
C08071=2778,29109,-32190,852,-26507,-1845
C08072=2776,29124,-32173,852,-26512,-1844
C08073=2775,29138,-32156,852,-26517,-1844
C08074=2764,29147,-32145,853,-26521,-1839
C08075=2763,29161,-32128,853,-26526,-1839
C08076=2763,29161,-30728,853,-26526,-1839
C08077=2904,29117,-28180,833,-26511,-1894
C08078=2904,29117,-32180,833,-26511,-1894
C08079=2911,29113,-32186,832,-26509,-1896
C08080=2915,29106,-32194,832,-26507,-1898
C08081=2915,29098,-32203,832,-26504,-1898
C08082=2916,29090,-32213,832,-26501,-1898
C08083=2917,29082,-32223,832,-26498,-1899
C08084=2917,29074,-32232,831,-26495,-1899
C08085=2918,29067,-32242,831,-26492,-1899
C08086=2919,29059,-32251,831,-26489,-1900
C08087=2920,29051,-32261,831,-26486,-1900
C08088=2919,29043,-32270,832,-26483,-1900
C08089=2913,29036,-32278,832,-26481,-1898
C08090=2911,29029,-32287,833,-26478,-1897
C08091=2912,29021,-32296,833,-26475,-1897
C08092=2912,29013,-32306,833,-26472,-1898
C08093=2913,29005,-32316,833,-26469,-1898
C08094=2914,28997,-32325,833,-26466,-1898
C08095=2914,28989,-32335,833,-26463,-1899
C08096=2915,28982,-32344,833,-26460,-1899
C08097=2913,28974,-32353,833,-26458,-1898
C08098=2908,28968,-32361,834,-26455,-1896
C08099=2907,28960,-32370,834,-26452,-1896
C08100=2907,28952,-32380,834,-26450,-1896
C08101=2908,28944,-32390,834,-26447,-1896
C08102=2909,28936,-32399,834,-26444,-1897
C08103=2909,28928,-32409,834,-26441,-1897
C08104=2910,28920,-32418,834,-26438,-1897
C08105=2911,28912,-32428,834,-26435,-1898
C08106=2912,28905,-32438,834,-26432,-1898
C08107=2909,28899,-32444,835,-26430,-1897
C08108=2900,28898,-32446,836,-26429,-1894
C08109=2891,28897,-32447,837,-26429,-1890
C08110=2890,28905,-32438,837,-26432,-1890
C08111=2890,28912,-32428,837,-26435,-1890
C08112=2889,28920,-32418,837,-26438,-1889
C08113=2888,28928,-32409,837,-26441,-1889
C08114=2888,28936,-32399,837,-26443,-1889
C08115=2887,28944,-32390,837,-26446,-1888
C08116=2893,28951,-32382,836,-26449,-1891
C08117=2896,28958,-32373,836,-26451,-1892
C08118=2896,28966,-32364,836,-26454,-1891
C08119=2895,28974,-32354,836,-26457,-1891
C08120=2894,28982,-32345,836,-26460,-1891
C08121=2893,28989,-32335,836,-26463,-1890
C08122=2893,28997,-32325,836,-26466,-1890
C08123=2892,29005,-32316,836,-26469,-1890
C08124=2891,29013,-32306,836,-26472,-1889
C08125=2891,29021,-32297,836,-26475,-1889
C08126=2897,29028,-32289,835,-26477,-1891
C08127=2900,29035,-32280,835,-26480,-1893
C08128=2899,29043,-32271,835,-26483,-1892
C08129=2898,29051,-32261,835,-26486,-1892
C08130=2898,29059,-32251,835,-26489,-1892
C08131=2902,29065,-32243,834,-26491,-1893
C08132=2907,29072,-32235,833,-26494,-1895
C08133=2906,29080,-32226,833,-26497,-1895
C08134=2906,29088,-32216,833,-26500,-1894
C08135=2905,29096,-32206,833,-26503,-1894
C08136=2904,29104,-32197,833,-26506,-1894
C08137=2904,29112,-32187,833,-26509,-1893
C08138=2904,29117,-32180,833,-26511,-1894
C08139=2904,29117,-30780,833,-26511,-1894
C08140=2896,28840,-28516,837,-26408,-1893
C08141=2896,28840,-32516,837,-26408,-1893
C08142=2905,28834,-32523,836,-26406,-1896
C08143=2908,28824,-32535,836,-26402,-1897
C08144=2909,28813,-32548,836,-26398,-1898
C08145=2910,28802,-32561,835,-26394,-1898
C08146=2911,28792,-32574,835,-26390,-1899
C08147=2909,28782,-32586,836,-26386,-1898
C08148=2902,28773,-32597,837,-26383,-1895
C08149=2901,28762,-32610,837,-26379,-1895
C08150=2893,28753,-32620,838,-26376,-1892
C08151=2893,28743,-32633,839,-26372,-1892
C08152=2885,28734,-32644,840,-26369,-1889
C08153=2878,28725,-32654,841,-26365,-1886
C08154=2876,28715,-32666,842,-26362,-1886
C08155=2876,28705,-32679,842,-26358,-1886
C08156=2877,28694,-32692,841,-26354,-1886
C08157=2878,28683,-32705,841,-26350,-1887
C08158=2879,28672,-32718,841,-26346,-1887
C08159=2880,28662,-32731,841,-26342,-1888
C08160=2881,28651,-32744,841,-26338,-1888
C08161=2887,28643,-32754,841,-26335,-1891
C08162=2893,28635,-32764,840,-26332,-1893
C08163=2894,28624,-32777,840,-26328,-1893
C08164=2900,28616,-32786,839,-26325,-1896
C08165=2906,28608,-32796,838,-26322,-1898
C08166=2907,28597,-32809,838,-26318,-1899
C08167=2913,28589,-32819,837,-26315,-1901
C08168=2919,28581,-32828,837,-26312,-1903
C08169=2924,28573,-32839,836,-26309,-1905
C08170=2929,28566,-32847,835,-26307,-1907
C08171=2921,28557,-32858,836,-26303,-1904
C08172=2919,28567,-32846,837,-26307,-1904
C08173=2910,28573,-32838,838,-26309,-1900
C08174=2908,28584,-32826,838,-26313,-1899
C08175=2899,28590,-32818,839,-26315,-1896
C08176=2896,28600,-32806,840,-26319,-1894
C08177=2888,28607,-32798,841,-26321,-1891
C08178=2884,28616,-32787,841,-26325,-1890
C08179=2877,28623,-32778,842,-26328,-1887
C08180=2872,28632,-32767,843,-26331,-1885
C08181=2871,28643,-32754,843,-26335,-1884
C08182=2864,28650,-32745,844,-26337,-1882
C08183=2859,28659,-32735,845,-26341,-1880
C08184=2858,28669,-32722,845,-26344,-1879
C08185=2857,28680,-32709,845,-26348,-1879
C08186=2857,28691,-32696,845,-26352,-1878
C08187=2856,28702,-32683,845,-26356,-1878
C08188=2855,28712,-32670,845,-26360,-1877
C08189=2857,28722,-32658,844,-26364,-1878
C08190=2864,28731,-32647,843,-26367,-1881
C08191=2865,28742,-32635,843,-26371,-1881
C08192=2872,28750,-32624,842,-26375,-1884
C08193=2880,28759,-32613,840,-26378,-1887
C08194=2888,28768,-32603,839,-26381,-1890
C08195=2891,28778,-32591,839,-26385,-1891
C08196=2896,28787,-32579,838,-26388,-1893
C08197=2900,28797,-32568,837,-26392,-1894
C08198=2899,28808,-32555,837,-26396,-1894
C08199=2898,28818,-32542,837,-26400,-1893
C08200=2897,28829,-32529,837,-26404,-1893
C08201=2896,28840,-32516,837,-26408,-1893
C08202=2896,28840,-31116,837,-26408,-1893
C08203=2469,28912,-28430,900,-26432,-1727
C08204=2469,28912,-32430,900,-26432,-1727
C08205=2444,28952,-32382,903,-26446,-1717
C08206=2406,28984,-32344,908,-26458,-1702
C08207=2359,29002,-32322,915,-26464,-1684
C08208=2311,29014,-32308,922,-26468,-1665
C08209=2262,29024,-32296,929,-26471,-1646
C08210=2215,29038,-32279,936,-26476,-1628
C08211=2163,29041,-32275,943,-26477,-1608
C08212=2115,29052,-32262,950,-26481,-1589
C08213=2063,29054,-32260,958,-26481,-1569
C08214=2012,29060,-32253,965,-26483,-1549
C08215=1966,29076,-32234,972,-26488,-1531
C08216=1919,29091,-32215,979,-26494,-1513
C08217=1870,29103,-32202,985,-26498,-1494
C08218=1820,29109,-32195,993,-26500,-1475
C08219=1771,29117,-32185,1000,-26502,-1456
C08220=1719,29119,-32182,1008,-26503,-1436
C08221=1668,29122,-32180,1015,-26503,-1416
C08222=1616,29124,-32178,1023,-26503,-1396
C08223=1564,29126,-32175,1030,-26504,-1376
C08224=1513,29128,-30773,1038,-26504,-1356
C08225=-41004,59868,4099,4900,-34257,16705
C08226=-41004,59868,1099,4900,-34257,16705
C08227=-41004,64596,1380,5213,-31659,16463
C08228=-41004,59868,1099,4900,-34257,16705
C08229=-41004,59868,9099,4900,-34257,16705
C08230=1513,29128,-28173,1038,-26504,-1356
C08231=1513,29128,-32173,1038,-26504,-1356
C08232=1463,29134,-32166,1045,-26506,-1336
C08233=1415,29123,-32179,1052,-26502,-1318
C08234=1369,29098,-32210,1059,-26492,-1300
C08235=1319,29081,-32231,1067,-26485,-1281
C08236=1264,29073,-32241,1075,-26482,-1260
C08237=1216,29085,-32226,1082,-26486,-1241
C08238=1165,29089,-32222,1089,-26487,-1222
C08239=1117,29099,-32209,1096,-26491,-1203
C08240=1065,29101,-32207,1104,-26491,-1183
C08241=1061,29110,-32196,1104,-26494,-1181
C08242=1113,29109,-32198,1097,-26494,-1201
C08243=1164,29106,-32201,1089,-26494,-1221
C08244=1216,29104,-32203,1082,-26493,-1241
C08245=1263,29092,-32218,1075,-26489,-1260
C08246=1315,29090,-32220,1067,-26489,-1279
C08247=1365,29107,-32199,1060,-26496,-1299
C08248=1406,29141,-32158,1053,-26508,-1314
C08249=1452,29148,-32149,1046,-26511,-1332
C08250=1505,29148,-32148,1039,-26512,-1352
C08251=1555,29144,-32154,1031,-26510,-1372
C08252=1607,29141,-32156,1024,-26510,-1392
C08253=1658,29139,-32159,1016,-26510,-1412
C08254=1710,29137,-32161,1009,-26509,-1432
C08255=1762,29135,-32163,1001,-26509,-1452
C08256=1813,29132,-32167,994,-26508,-1472
C08257=1861,29121,-32180,987,-26504,-1491
C08258=1913,29119,-32182,979,-26504,-1510
C08259=1958,29099,-32206,973,-26497,-1528
C08260=2006,29084,-32224,966,-26492,-1547
C08261=2054,29072,-32238,959,-26488,-1565
C08262=2105,29070,-32241,951,-26487,-1585
C08263=2156,29064,-32247,944,-26486,-1605
C08264=2208,29063,-32249,936,-26485,-1625
C08265=2255,29047,-32268,930,-26480,-1643
C08266=2302,29031,-32286,923,-26475,-1662
C08267=2351,29022,-32297,916,-26472,-1681
C08268=2398,29007,-32316,909,-26466,-1699
C08269=2443,28984,-32343,903,-26458,-1716
C08270=2476,28955,-32379,898,-26447,-1729
C08271=2469,28912,-32430,900,-26432,-1727
C08272=2469,28912,-31030,900,-26432,-1727
C08273=2271,28794,-28573,930,-26387,-1652
C08274=2271,28794,-32573,930,-26387,-1652
C08275=2279,28785,-32584,929,-26383,-1655
C08276=2286,28775,-32596,928,-26380,-1657
C08277=2296,28768,-32605,927,-26377,-1661
C08278=2302,28758,-32617,926,-26373,-1664
C08279=2292,28753,-32623,927,-26372,-1660
C08280=2281,28761,-32614,929,-26374,-1656
C08281=2278,28772,-32600,929,-26378,-1654
C08282=2267,28780,-32591,931,-26381,-1650
C08283=2257,28787,-32582,932,-26384,-1646
C08284=2246,28794,-32573,934,-26386,-1642
C08285=2233,28795,-32572,936,-26387,-1637
C08286=2222,28803,-32563,937,-26389,-1633
C08287=2211,28808,-32557,939,-26391,-1628
C08288=2198,28811,-32553,941,-26392,-1623
C08289=2186,28814,-32549,942,-26393,-1618
C08290=2174,28819,-32544,944,-26395,-1614
C08291=2164,28827,-32534,946,-26398,-1610
C08292=2153,28834,-32525,947,-26401,-1606
C08293=2140,28836,-32523,949,-26401,-1601
C08294=2129,28842,-32516,950,-26403,-1596
C08295=2119,28850,-32506,952,-26406,-1592
C08296=2105,28850,-32506,954,-26406,-1587
C08297=2095,28858,-32497,955,-26409,-1583
C08298=2082,28858,-32496,957,-26409,-1578
C08299=2071,28866,-32487,959,-26412,-1574
C08300=2060,28872,-32480,960,-26414,-1569
C08301=2047,28874,-32477,962,-26415,-1564
C08302=2035,28878,-32472,964,-26416,-1560
C08303=2023,28882,-32468,966,-26417,-1555
C08304=2013,28890,-32458,967,-26420,-1551
C08305=2000,28892,-32455,969,-26421,-1546
C08306=1989,28898,-32449,970,-26423,-1542
C08307=1985,28909,-32435,971,-26427,-1540
C08308=1985,28922,-32420,971,-26432,-1540
C08309=1990,28924,-32417,970,-26433,-1542
C08310=1996,28914,-32429,969,-26429,-1544
C08311=2004,28905,-32440,968,-26426,-1547
C08312=2017,28904,-32441,966,-26426,-1552
C08313=2027,28897,-32450,965,-26423,-1557
C08314=2041,28897,-32450,963,-26423,-1562
C08315=2052,28890,-32458,961,-26421,-1566
C08316=2064,28889,-32460,959,-26420,-1571
C08317=2075,28881,-32469,958,-26417,-1575
C08318=2087,28876,-32475,956,-26416,-1580
C08319=2099,28873,-32479,955,-26414,-1584
C08320=2111,28870,-32482,953,-26414,-1589
C08321=2123,28865,-32488,951,-26412,-1594
C08322=2133,28857,-32497,950,-26409,-1598
C08323=2146,28856,-32499,948,-26409,-1603
C08324=2157,28849,-32507,946,-26406,-1607
C08325=2168,28842,-32516,945,-26403,-1611
C08326=2178,28834,-32525,943,-26401,-1615
C08327=2192,28833,-32526,941,-26401,-1621
C08328=2202,28826,-32535,940,-26398,-1625
C08329=2215,28825,-32536,938,-26398,-1630
C08330=2226,28818,-32545,936,-26395,-1634
C08331=2237,28812,-32552,935,-26393,-1638
C08332=2250,28810,-32555,933,-26392,-1643
C08333=2261,28802,-32564,932,-26389,-1647
C08334=2271,28794,-32573,930,-26387,-1652
C08335=2271,28794,-31173,930,-26387,-1652
C08336=1994,28765,-28609,971,-26374,-1545
C08337=1994,28765,-32609,971,-26374,-1545
C08338=1987,28758,-32618,972,-26371,-1542
C08339=1981,28750,-32628,974,-26368,-1540
C08340=1972,28745,-32634,975,-26366,-1536
C08341=1962,28744,-32635,976,-26366,-1532
C08342=1953,28739,-32641,978,-26364,-1529
C08343=1946,28732,-32650,979,-26361,-1526
C08344=1936,28730,-32652,980,-26360,-1522
C08345=1929,28722,-32661,981,-26358,-1520
C08346=1920,28718,-32666,983,-26356,-1516
C08347=1909,28717,-32668,984,-26356,-1512
C08348=1901,28711,-32675,986,-26353,-1509
C08349=1893,28705,-32682,987,-26351,-1506
C08350=1883,28704,-32684,988,-26350,-1502
C08351=1872,28702,-32686,990,-26350,-1498
C08352=1862,28701,-32688,992,-26349,-1494
C08353=1852,28698,-32691,993,-26348,-1491
C08354=1846,28690,-32701,994,-26345,-1488
C08355=1836,28687,-32704,996,-26344,-1484
C08356=1825,28686,-32706,997,-26343,-1480
C08357=1815,28684,-32708,999,-26343,-1476
C08358=1807,28678,-32716,1000,-26340,-1473
C08359=1799,28672,-32722,1001,-26338,-1470
C08360=1789,28671,-32724,1003,-26338,-1466
C08361=1778,28669,-32726,1004,-26337,-1462
C08362=1769,28665,-32731,1006,-26335,-1459
C08363=1762,28658,-32740,1007,-26333,-1456
C08364=1752,28656,-32742,1008,-26332,-1452
C08365=1742,28654,-32744,1010,-26331,-1448
C08366=1731,28653,-32746,1012,-26331,-1444
C08367=1730,28662,-32734,1012,-26334,-1444
C08368=1737,28670,-32725,1010,-26337,-1446
C08369=1746,28674,-32720,1009,-26339,-1450
C08370=1757,28676,-32718,1007,-26339,-1454
C08371=1767,28677,-32716,1006,-26340,-1458
C08372=1775,28682,-32710,1005,-26342,-1461
C08373=1783,28689,-32702,1003,-26344,-1464
C08374=1793,28691,-32700,1002,-26345,-1468
C08375=1804,28692,-32698,1000,-26346,-1472
C08376=1814,28695,-32695,999,-26347,-1476
C08377=1821,28702,-32686,998,-26350,-1478
C08378=1830,28705,-32682,996,-26351,-1482
C08379=1841,28707,-32680,995,-26351,-1486
C08380=1851,28708,-32678,993,-26352,-1490
C08381=1859,28715,-32671,992,-26354,-1493
C08382=1867,28720,-32664,991,-26356,-1496
C08383=1877,28722,-32662,989,-26357,-1500
C08384=1888,28723,-32660,988,-26358,-1504
C08385=1897,28727,-32656,986,-26359,-1507
C08386=1904,28735,-32646,985,-26362,-1510
C08387=1914,28737,-32644,984,-26363,-1514
C08388=1924,28738,-32642,982,-26363,-1518
C08389=1931,28746,-32633,981,-26366,-1521
C08390=1940,28750,-32628,979,-26368,-1524
C08391=1950,28751,-32626,978,-26369,-1528
C08392=1959,28756,-32620,977,-26370,-1531
C08393=1966,28763,-32612,975,-26373,-1534
C08394=1976,28766,-32609,974,-26374,-1538
C08395=1983,28773,-32599,973,-26377,-1540
C08396=1991,28772,-32601,972,-26376,-1543
C08397=1994,28765,-31209,971,-26374,-1545
C08398=-41004,59868,4099,4900,-34257,16705
C08399=-41004,59868,1099,4900,-34257,16705
C08400=-41004,64596,1380,5213,-31659,16463
C08401=-41004,59868,1099,4900,-34257,16705
C08402=-41004,59868,9099,4900,-34257,16705
C08403=1994,28765,-28609,971,-26374,-1545
C08404=1994,28765,-32609,971,-26374,-1545
C08405=1994,28765,-31209,971,-26374,-1545
C08406=1471,28809,-28558,1048,-26386,-1342
C08407=1471,28809,-32558,1048,-26386,-1342
C08408=1429,28752,-32627,1055,-26365,-1327
C08409=1373,28709,-32679,1064,-26349,-1305
C08410=1313,28673,-32724,1073,-26335,-1282
C08411=1253,28636,-32768,1082,-26321,-1260
C08412=1199,28592,-32821,1091,-26305,-1239
C08413=1203,28533,-32893,1091,-26283,-1241
C08414=1234,28479,-32957,1087,-26263,-1254
C08415=1308,28487,-32948,1076,-26266,-1282
C08416=1377,28507,-32924,1066,-26274,-1309
C08417=1439,28503,-32927,1057,-26273,-1332
C08418=1482,28456,-32984,1051,-26256,-1349
C08419=1486,28388,-33066,1051,-26231,-1352
C08420=1475,28324,-33143,1054,-26208,-1348
C08421=1495,28275,-33203,1051,-26190,-1356
C08422=1569,28286,-33189,1040,-26194,-1385
C08423=1628,28251,-33231,1032,-26182,-1408
C08424=1670,28203,-33289,1026,-26164,-1424
C08425=1738,28195,-33298,1016,-26162,-1451
C08426=1767,28180,-33316,1012,-26157,-1462
C08427=1692,28170,-33329,1023,-26152,-1433
C08428=1640,28207,-33285,1031,-26165,-1413
C08429=1591,28251,-33232,1037,-26181,-1393
C08430=1528,28251,-33231,1047,-26181,-1369
C08431=1463,28258,-33224,1056,-26183,-1344
C08432=1459,28325,-33142,1056,-26208,-1342
C08433=1465,28390,-33064,1054,-26232,-1344
C08434=1456,28455,-32985,1055,-26256,-1339
C08435=1404,28491,-32942,1062,-26269,-1319
C08436=1334,28472,-32966,1072,-26261,-1292
C08437=1259,28461,-32979,1084,-26257,-1264
C08438=1206,28485,-32950,1091,-26265,-1243
C08439=1162,28532,-32894,1097,-26282,-1225
C08440=1098,28503,-32929,1107,-26271,-1201
C08441=1032,28476,-32962,1117,-26260,-1176
C08442=964,28455,-32988,1127,-26252,-1149
C08443=896,28430,-33017,1138,-26243,-1124
C08444=823,28417,-33033,1149,-26237,-1096
C08445=749,28406,-33047,1160,-26233,-1067
C08446=674,28396,-33060,1171,-26228,-1038
C08447=599,28385,-33073,1182,-26224,-1009
C08448=642,28410,-33043,1176,-26233,-1025
C08449=716,28421,-33029,1164,-26238,-1054
C08450=791,28432,-33016,1153,-26242,-1083
C08451=861,28451,-32992,1143,-26250,-1110
C08452=931,28469,-32971,1132,-26257,-1137
C08453=1005,28481,-32955,1121,-26262,-1165
C08454=1069,28510,-32921,1111,-26273,-1190
C08455=1132,28542,-32882,1101,-26285,-1214
C08456=1178,28587,-32827,1094,-26302,-1231
C08457=1227,28637,-32767,1086,-26321,-1249
C08458=1286,28675,-32721,1077,-26336,-1272
C08459=1346,28712,-32676,1068,-26350,-1295
C08460=1403,28753,-32626,1059,-26365,-1317
C08461=1448,28804,-32564,1051,-26384,-1334
C08462=1454,28862,-32494,1050,-26406,-1335
C08463=1412,28910,-32437,1055,-26423,-1319
C08464=1365,28943,-32397,1062,-26435,-1300
C08465=1424,28919,-32426,1053,-26427,-1323
C08466=1473,28875,-32479,1047,-26411,-1342
C08467=1471,28809,-32558,1048,-26386,-1342
C08468=1471,28809,-31158,1048,-26386,-1342
C08469=677,28906,-28444,1164,-26416,-1034
C08470=677,28906,-32444,1164,-26416,-1034
C08471=669,28901,-32450,1165,-26414,-1031
C08472=656,28899,-32453,1167,-26414,-1026
C08473=656,28911,-32439,1167,-26418,-1026
C08474=655,28922,-32425,1167,-26422,-1026
C08475=654,28933,-32411,1166,-26426,-1025
C08476=648,28942,-32401,1167,-26429,-1023
C08477=643,28951,-32391,1168,-26432,-1021
C08478=642,28962,-32377,1168,-26437,-1020
C08479=642,28973,-32363,1168,-26441,-1020
C08480=632,28980,-32355,1169,-26443,-1016
C08481=630,28991,-32342,1169,-26447,-1015
C08482=630,29002,-32328,1169,-26451,-1015
C08483=629,29014,-32315,1169,-26455,-1015
C08484=628,29025,-32301,1169,-26460,-1014
C08485=628,29036,-32287,1169,-26464,-1014
C08486=620,29044,-32278,1170,-26467,-1011
C08487=616,29054,-32266,1170,-26470,-1009
C08488=616,29065,-32253,1170,-26474,-1009
C08489=615,29077,-32239,1170,-26478,-1009
C08490=614,29088,-32225,1170,-26483,-1008
C08491=614,29099,-32211,1170,-26487,-1008
C08492=613,29111,-32198,1170,-26491,-1008
C08493=605,29118,-32189,1171,-26494,-1005
C08494=602,29128,-32177,1172,-26497,-1003
C08495=601,29139,-32163,1171,-26502,-1003
C08496=600,29151,-32149,1171,-26506,-1002
C08497=600,29162,-32136,1171,-26510,-1002
C08498=599,29174,-32122,1171,-26514,-1002
C08499=598,29185,-32108,1171,-26518,-1001
C08500=598,29196,-32094,1171,-26522,-1001
C08501=599,29205,-32085,1171,-26525,-1001
C08502=608,29198,-32093,1170,-26523,-1005
C08503=617,29191,-32101,1168,-26521,-1009
C08504=619,29180,-32114,1168,-26517,-1010
C08505=620,29169,-32127,1168,-26513,-1010
C08506=621,29158,-32141,1168,-26508,-1010
C08507=621,29146,-32155,1168,-26504,-1011
C08508=622,29135,-32168,1168,-26500,-1011
C08509=623,29123,-32182,1169,-26496,-1011
C08510=623,29112,-32196,1169,-26492,-1012
C08511=627,29102,-32208,1168,-26488,-1013
C08512=635,29095,-32217,1167,-26485,-1016
C08513=635,29083,-32231,1167,-26481,-1017
C08514=636,29072,-32244,1167,-26477,-1017
C08515=637,29061,-32258,1167,-26473,-1017
C08516=637,29049,-32272,1167,-26469,-1018
C08517=639,29039,-32285,1167,-26465,-1019
C08518=649,29032,-32293,1166,-26462,-1022
C08519=649,29020,-32306,1166,-26458,-1023
C08520=650,29009,-32320,1166,-26454,-1023
C08521=651,28998,-32334,1166,-26450,-1023
C08522=657,28989,-32344,1165,-26447,-1026
C08523=662,28980,-32355,1165,-26443,-1028
C08524=663,28969,-32368,1165,-26439,-1028
C08525=663,28958,-32382,1165,-26435,-1029
C08526=664,28946,-32396,1165,-26431,-1029
C08527=668,28936,-32408,1165,-26427,-1030
C08528=676,28929,-32417,1163,-26425,-1034
C08529=676,28917,-32431,1164,-26420,-1034
C08530=677,28906,-32444,1164,-26416,-1034
C08531=677,28906,-31044,1164,-26416,-1034
C08532=739,28185,-29313,1164,-26152,-1065
C08533=739,28185,-33313,1164,-26152,-1065
C08534=748,28179,-33320,1163,-26149,-1068
C08535=756,28174,-33328,1162,-26147,-1072
C08536=762,28166,-33336,1161,-26145,-1074
C08537=765,28158,-33347,1161,-26141,-1075
C08538=773,28152,-33354,1160,-26139,-1079
C08539=774,28142,-33366,1160,-26136,-1079
C08540=783,28136,-33373,1159,-26134,-1082
C08541=791,28130,-33380,1157,-26131,-1086
C08542=796,28122,-33389,1157,-26129,-1088
C08543=800,28114,-33399,1156,-26126,-1089
C08544=807,28108,-33407,1155,-26123,-1092
C08545=809,28098,-33418,1155,-26120,-1093
C08546=818,28092,-33425,1154,-26118,-1096
C08547=819,28083,-33437,1154,-26114,-1097
C08548=827,28077,-33444,1153,-26112,-1100
C08549=835,28071,-33451,1152,-26110,-1103
C08550=841,28064,-33460,1151,-26107,-1106
C08551=845,28055,-33470,1150,-26104,-1107
C08552=853,28049,-33478,1149,-26102,-1110
C08553=854,28039,-33489,1149,-26098,-1111
C08554=862,28033,-33497,1148,-26096,-1114
C08555=870,28027,-33504,1147,-26094,-1117
C08556=876,28020,-33513,1146,-26091,-1119
C08557=880,28012,-33523,1146,-26088,-1121
C08558=887,28005,-33530,1145,-26086,-1124
C08559=889,27996,-33542,1145,-26083,-1125
C08560=897,27990,-33549,1144,-26081,-1128
C08561=899,27980,-33560,1143,-26077,-1129
C08562=900,27970,-33572,1143,-26073,-1129
C08563=901,27960,-33584,1143,-26070,-1130
C08564=892,27966,-33577,1145,-26072,-1126
C08565=889,27975,-33567,1145,-26075,-1125
C08566=883,27982,-33558,1146,-26078,-1123
C08567=875,27988,-33551,1147,-26080,-1119
C08568=867,27994,-33544,1148,-26082,-1116
C08569=865,28004,-33532,1148,-26086,-1116
C08570=857,28010,-33525,1149,-26088,-1112
C08571=855,28019,-33514,1149,-26091,-1111
C08572=848,28026,-33506,1150,-26093,-1109
C08573=839,28032,-32099,1152,-26096,-1105
C08574=-41004,59868,4099,4900,-34257,16705
C08575=-41004,59868,1099,4900,-34257,16705
C08576=-41004,64596,1380,5213,-31659,16463
C08577=-41004,59868,1099,4900,-34257,16705
C08578=-41004,59868,9099,4900,-34257,16705
C08579=839,28032,-29499,1152,-26096,-1105
C08580=839,28032,-33499,1152,-26096,-1105
C08581=832,28038,-33491,1152,-26098,-1103
C08582=830,28047,-33480,1153,-26101,-1102
C08583=822,28053,-33472,1154,-26103,-1098
C08584=820,28063,-33461,1154,-26107,-1098
C08585=813,28069,-33453,1155,-26109,-1095
C08586=804,28075,-33446,1156,-26111,-1091
C08587=798,28082,-33438,1157,-26114,-1089
C08588=795,28091,-33427,1157,-26117,-1088
C08589=787,28097,-33420,1158,-26119,-1084
C08590=786,28107,-33408,1158,-26123,-1084
C08591=777,28113,-33401,1160,-26125,-1081
C08592=775,28121,-33390,1160,-26128,-1079
C08593=768,28128,-33382,1161,-26131,-1077
C08594=760,28134,-33375,1162,-26133,-1074
C08595=752,28141,-33367,1163,-26135,-1071
C08596=751,28150,-33356,1163,-26139,-1070
C08597=742,28156,-33349,1164,-26141,-1067
C08598=740,28165,-33338,1164,-26144,-1066
C08599=740,28175,-33325,1164,-26148,-1066
C08600=739,28185,-33313,1164,-26152,-1065
C08601=739,28185,-31913,1164,-26152,-1065
C08602=3144,28439,-29000,805,-26261,-1991
C08603=3144,28439,-33000,805,-26261,-1991
C08604=3154,28447,-32990,803,-26264,-1995
C08605=3172,28449,-32987,800,-26265,-2002
C08606=3189,28452,-32984,798,-26266,-2009
C08607=3207,28454,-32982,795,-26267,-2015
C08608=3222,28447,-32990,793,-26265,-2021
C08609=3239,28450,-32987,790,-26266,-2028
C08610=3255,28447,-32990,788,-26265,-2034
C08611=3272,28445,-32992,786,-26264,-2040
C08612=3289,28447,-32989,783,-26265,-2047
C08613=3304,28440,-32998,781,-26262,-2053
C08614=3321,28442,-32995,778,-26263,-2060
C08615=3339,28445,-32992,776,-26264,-2066
C08616=3357,28447,-32989,773,-26266,-2073
C08617=3372,28455,-32979,771,-26269,-2079
C08618=3375,28470,-32961,770,-26274,-2080
C08619=3373,28486,-32942,770,-26280,-2079
C08620=3376,28501,-32924,770,-26286,-2080
C08621=3381,28516,-32906,769,-26291,-2082
C08622=3391,28529,-32890,767,-26296,-2086
C08623=3406,28536,-32881,765,-26299,-2092
C08624=3422,28543,-32873,762,-26301,-2097
C08625=3437,28550,-32864,760,-26304,-2103
C08626=3449,28549,-32866,758,-26304,-2108
C08627=3466,28549,-32866,756,-26304,-2115
C08628=3484,28551,-32863,753,-26305,-2121
C08629=3499,28544,-32871,751,-26302,-2127
C08630=3514,28539,-32877,749,-26301,-2133
C08631=3527,28530,-32889,747,-26297,-2138
C08632=3540,28520,-32901,745,-26293,-2143
C08633=3548,28507,-32916,744,-26289,-2146
C08634=3564,28506,-32918,742,-26289,-2153
C08635=3574,28499,-32926,740,-26286,-2156
C08636=3563,28486,-32942,742,-26281,-2152
C08637=3550,28475,-32955,744,-26277,-2147
C08638=3537,28465,-32967,746,-26273,-2142
C08639=3520,28461,-32972,749,-26272,-2136
C08640=3502,28458,-32976,751,-26270,-2129
C08641=3489,28447,-32989,753,-26266,-2124
C08642=3472,28445,-32992,756,-26265,-2117
C08643=3454,28442,-32995,759,-26264,-2111
C08644=3436,28440,-32998,761,-26263,-2104
C08645=3418,28437,-33001,764,-26262,-2097
C08646=3400,28434,-33004,767,-26261,-2090
C08647=3383,28432,-33008,769,-26260,-2083
C08648=3365,28429,-33011,772,-26259,-2076
C08649=3347,28427,-33014,775,-26258,-2069
C08650=3333,28434,-33005,777,-26261,-2064
C08651=3315,28432,-33008,779,-26259,-2057
C08652=3297,28429,-33011,782,-26258,-2050
C08653=3280,28429,-33011,785,-26258,-2044
C08654=3265,28434,-33005,787,-26260,-2038
C08655=3247,28432,-33008,789,-26259,-2031
C08656=3229,28429,-33011,792,-26258,-2024
C08657=3215,28436,-33002,794,-26261,-2018
C08658=3201,28427,-33014,796,-26257,-2013
C08659=3196,28415,-33029,797,-26252,-2011
C08660=3178,28412,-33032,800,-26251,-2004
C08661=3164,28420,-33023,802,-26254,-1999
C08662=3148,28424,-33018,804,-26256,-1993
C08663=3144,28439,-33000,805,-26261,-1991
C08664=3144,28439,-31600,805,-26261,-1991
C08665=3243,28517,-28905,789,-26291,-2029
C08666=3243,28517,-32905,789,-26291,-2029
C08667=3242,28525,-32896,789,-26293,-2028
C08668=3246,28531,-32888,788,-26296,-2030
C08669=3252,28538,-32880,788,-26298,-2032
C08670=3257,28544,-32872,787,-26301,-2034
C08671=3264,28549,-32867,786,-26302,-2037
C08672=3272,28551,-32864,784,-26303,-2040
C08673=3278,28557,-32857,784,-26306,-2042
C08674=3285,28561,-32851,783,-26307,-2044
C08675=3293,28563,-32849,781,-26308,-2048
C08676=3298,28570,-32841,780,-26310,-2050
C08677=3305,28574,-32836,779,-26312,-2052
C08678=3313,28576,-32833,778,-26313,-2055
C08679=3319,28582,-32826,777,-26315,-2057
C08680=3326,28586,-32821,776,-26317,-2060
C08681=3334,28588,-32820,775,-26317,-2063
C08682=3343,28589,-32818,774,-26318,-2067
C08683=3348,28595,-32810,773,-26320,-2069
C08684=3355,28600,-32804,772,-26322,-2071
C08685=3363,28601,-32803,770,-26323,-2075
C08686=3372,28602,-32801,769,-26323,-2078
C08687=3380,28604,-32800,768,-26324,-2081
C08688=3387,28608,-32794,767,-26325,-2084
C08689=3392,28615,-32786,766,-26328,-2086
C08690=3401,28616,-32785,765,-26328,-2089
C08691=3409,28617,-32783,763,-26329,-2092
C08692=3418,28619,-32782,762,-26329,-2096
C08693=3426,28618,-32782,761,-26329,-2099
C08694=3433,28614,-32788,760,-26328,-2101
C08695=3440,28612,-32789,759,-26327,-2104
C08696=3448,28612,-32790,758,-26327,-2107
C08697=3455,28607,-32796,757,-26325,-2110
C08698=3452,28604,-32799,757,-26324,-2109
C08699=3443,28603,-32800,759,-26324,-2105
C08700=3435,28602,-32802,760,-26323,-2102
C08701=3426,28601,-32803,761,-26323,-2099
C08702=3417,28600,-32805,762,-26322,-2095
C08703=3409,28598,-32806,764,-26322,-2092
C08704=3400,28597,-32808,765,-26321,-2089
C08705=3392,28596,-32809,766,-26321,-2086
C08706=3383,28595,-32811,768,-26320,-2082
C08707=3375,28593,-32812,769,-26320,-2079
C08708=3369,28588,-32819,770,-26318,-2077
C08709=3363,28582,-32826,771,-26315,-2074
C08710=3354,28581,-32828,772,-26315,-2071
C08711=3346,28580,-32829,773,-26314,-2068
C08712=3337,28578,-32831,775,-26314,-2065
C08713=3330,28575,-32835,776,-26312,-2062
C08714=3324,28568,-32843,777,-26310,-2060
C08715=3316,28566,-32846,778,-26309,-2057
C08716=3310,28562,-32851,779,-26308,-2054
C08717=3304,28555,-32858,780,-26305,-2052
C08718=3296,28553,-32861,781,-26304,-2049
C08719=3289,28549,-32866,782,-26303,-2046
C08720=3284,28543,-32874,783,-26300,-2044
C08721=3275,28541,-32876,784,-26300,-2041
C08722=3269,28536,-32882,785,-26298,-2039
C08723=3263,28530,-32890,786,-26295,-2036
C08724=3258,28523,-32897,787,-26293,-2034
C08725=3251,28518,-32904,788,-26291,-2032
C08726=3243,28517,-32905,789,-26291,-2029
C08727=3243,28517,-31505,789,-26291,-2029
C08728=3847,28629,-28768,698,-26336,-2261
C08729=3847,28629,-32768,698,-26336,-2261
C08730=3845,28653,-32739,698,-26345,-2260
C08731=3843,28676,-32711,698,-26353,-2259
C08732=3857,28687,-32698,696,-26358,-2265
C08733=3865,28666,-32723,695,-26350,-2268
C08734=3867,28643,-32751,695,-26341,-2269
C08735=3870,28619,-32779,695,-26333,-2270
C08736=3882,28601,-32801,693,-26326,-2275
C08737=3885,28578,-32829,693,-26317,-2276
C08738=3897,28560,-32851,692,-26311,-2281
C08739=3905,28540,-32876,690,-26303,-2284
C08740=3918,28522,-32897,689,-26297,-2289
C08741=3931,28504,-32919,687,-26290,-2294
C08742=3944,28486,-32940,685,-26284,-2299
C08743=3957,28469,-32961,683,-26277,-2305
C08744=3978,28455,-32978,681,-26272,-2312
C08745=3998,28441,-32995,678,-26267,-2320
C08746=4020,28434,-33003,674,-26265,-2329
C08747=4043,28427,-33011,671,-26262,-2338
C08748=4065,28420,-33020,668,-26260,-2346
C08749=4090,28419,-31621,664,-26260,-2356
C08750=-41004,59868,4099,4900,-34257,16705
C08751=-41004,59868,1099,4900,-34257,16705
C08752=-41004,64596,1380,5213,-31659,16463
C08753=-41004,59868,1099,4900,-34257,16705
C08754=-41004,59868,9099,4900,-34257,16705
C08755=4090,28419,-29021,664,-26260,-2356
C08756=4090,28419,-33021,664,-26260,-2356
C08757=4112,28413,-33029,661,-26257,-2365
C08758=4139,28416,-33024,657,-26259,-2375
C08759=4165,28420,-33020,653,-26260,-2385
C08760=4191,28424,-33015,649,-26262,-2395
C08761=4217,28428,-33011,645,-26264,-2405
C08762=4242,28433,-33004,641,-26266,-2415
C08763=4264,28444,-32991,638,-26270,-2423
C08764=4290,28448,-32986,634,-26271,-2433
C08765=4316,28451,-32982,630,-26273,-2443
C08766=4337,28464,-32966,627,-26278,-2451
C08767=4363,28468,-32962,623,-26279,-2461
C08768=4386,28462,-32968,620,-26277,-2470
C08769=4367,28449,-32984,623,-26272,-2463
C08770=4341,28445,-32989,626,-26271,-2452
C08771=4318,28436,-33000,630,-26267,-2444
C08772=4294,28429,-33009,634,-26265,-2435
C08773=4268,28425,-33013,638,-26263,-2424
C08774=4247,28413,-33028,641,-26258,-2417
C08775=4221,28409,-33033,645,-26257,-2407
C08776=4195,28405,-33038,649,-26255,-2396
C08777=4169,28402,-33042,653,-26254,-2386
C08778=4143,28398,-33047,656,-26252,-2376
C08779=4117,28394,-33051,660,-26250,-2366
C08780=4094,28400,-33044,664,-26253,-2358
C08781=4069,28401,-33044,667,-26253,-2348
C08782=4046,28407,-33036,671,-26255,-2339
C08783=4024,28414,-33027,674,-26257,-2331
C08784=4001,28421,-33019,677,-26260,-2322
C08785=3979,28428,-33011,681,-26262,-2313
C08786=3959,28442,-32994,683,-26267,-2305
C08787=3940,28456,-32977,686,-26272,-2298
C08788=3927,28474,-32955,688,-26279,-2293
C08789=3915,28492,-32933,690,-26286,-2288
C08790=3902,28510,-32911,691,-26292,-2283
C08791=3890,28528,-32890,693,-26299,-2278
C08792=3881,28548,-32866,694,-26306,-2274
C08793=3868,28566,-32844,696,-26313,-2269
C08794=3862,28588,-32818,696,-26321,-2267
C08795=3860,28611,-32789,697,-26329,-2266
C08796=3847,28629,-32768,698,-26336,-2261
C08797=3847,28629,-31368,698,-26336,-2261
C08798=3979,28612,-28788,679,-26330,-2312
C08799=3979,28612,-32788,679,-26330,-2312
C08800=4013,28597,-32807,674,-26325,-2325
C08801=4048,28585,-32820,669,-26321,-2339
C08802=4086,28581,-32825,663,-26320,-2354
C08803=4121,28567,-32842,658,-26315,-2367
C08804=4158,28579,-32827,652,-26320,-2381
C08805=4168,28614,-32785,651,-26332,-2385
C08806=4188,28646,-32747,647,-26344,-2392
C08807=4220,28667,-32721,643,-26353,-2405
C08808=4258,28663,-32726,637,-26351,-2419
C08809=4296,28659,-32730,631,-26350,-2434
C08810=4331,28648,-32744,626,-26346,-2448
C08811=4358,28623,-32774,622,-26337,-2458
C08812=4393,28617,-32781,617,-26335,-2471
C08813=4427,28635,-32759,612,-26342,-2484
C08814=4463,28636,-32758,607,-26342,-2498
C08815=4504,28641,-32752,601,-26345,-2514
C08816=4541,28634,-32760,595,-26342,-2528
C08817=4575,28619,-32778,590,-26337,-2542
C08818=4577,28604,-32796,590,-26331,-2543
C08819=4540,28609,-32790,595,-26333,-2528
C08820=4506,28620,-32777,600,-26337,-2515
C08821=4474,28598,-32803,605,-26329,-2503
C08822=4438,28584,-32821,611,-26323,-2489
C08823=4407,28560,-32850,616,-26314,-2477
C08824=4371,28545,-32868,621,-26308,-2464
C08825=4335,28531,-32885,627,-26303,-2450
C08826=4299,28516,-32903,632,-26297,-2436
C08827=4258,28510,-32911,638,-26294,-2420
C08828=4222,28495,-32929,644,-26289,-2406
C08829=4181,28489,-32936,650,-26286,-2390
C08830=4139,28483,-32943,656,-26284,-2374
C08831=4101,28487,-32938,662,-26285,-2360
C08832=4063,28492,-32933,667,-26287,-2345
C08833=4036,28511,-32910,671,-26293,-2335
C08834=4036,28528,-32890,671,-26300,-2335
C08835=4070,28512,-32909,666,-26294,-2348
C08836=4105,28498,-32926,661,-26289,-2361
C08837=4147,28504,-32919,655,-26291,-2377
C08838=4188,28509,-32912,649,-26294,-2393
C08839=4229,28515,-32904,642,-26296,-2409
C08840=4271,28521,-32897,636,-26299,-2425
C08841=4309,28532,-32885,630,-26303,-2440
C08842=4347,28543,-32870,625,-26307,-2454
C08843=4381,28561,-32848,619,-26314,-2467
C08844=4413,28574,-32833,615,-26319,-2479
C08845=4436,28593,-32810,611,-26326,-2488
C08846=4444,28614,-32785,610,-26334,-2491
C08847=4411,28609,-32791,615,-26332,-2479
C08848=4370,28603,-32798,621,-26329,-2463
C08849=4332,28590,-32814,626,-26324,-2448
C08850=4292,28582,-32824,633,-26321,-2433
C08851=4256,28567,-32842,638,-26316,-2419
C08852=4215,28561,-32849,644,-26313,-2403
C08853=4173,28555,-32856,650,-26311,-2387
C08854=4135,28559,-32851,656,-26312,-2373
C08855=4095,28557,-32854,662,-26311,-2357
C08856=4059,28565,-32845,667,-26314,-2343
C08857=4021,28572,-32837,673,-26316,-2329
C08858=3985,28581,-32826,678,-26319,-2315
C08859=3979,28612,-32788,679,-26330,-2312
C08860=3979,28612,-31388,679,-26330,-2312
C08861=4084,28699,-28682,662,-26364,-2352
C08862=4084,28699,-32682,662,-26364,-2352
C08863=4086,28705,-32675,662,-26366,-2353
C08864=4095,28707,-32672,661,-26367,-2356
C08865=4101,28714,-32664,660,-26369,-2358
C08866=4109,28718,-32659,659,-26371,-2361
C08867=4118,28719,-32658,657,-26371,-2365
C08868=4126,28722,-32655,656,-26372,-2368
C08869=4132,28729,-32646,655,-26375,-2370
C08870=4140,28732,-32642,654,-26376,-2373
C08871=4149,28733,-32641,652,-26377,-2377
C08872=4158,28735,-32639,651,-26377,-2380
C08873=4167,28736,-32637,650,-26378,-2384
C08874=4176,28737,-32636,648,-26378,-2387
C08875=4185,28739,-32634,647,-26379,-2391
C08876=4193,28735,-32639,646,-26377,-2394
C08877=4200,28731,-32643,645,-26376,-2397
C08878=4209,28733,-32641,643,-26377,-2400
C08879=4219,28734,-32640,642,-26377,-2404
C08880=4226,28729,-32646,641,-26376,-2406
C08881=4233,28726,-32649,640,-26375,-2409
C08882=4243,28728,-32647,639,-26375,-2413
C08883=4252,28729,-32646,637,-26376,-2416
C08884=4259,28724,-32652,636,-26374,-2419
C08885=4267,28722,-32654,635,-26373,-2422
C08886=4276,28723,-32653,634,-26374,-2426
C08887=4285,28723,-32652,632,-26374,-2429
C08888=4292,28719,-32658,631,-26372,-2432
C08889=4300,28717,-32660,630,-26372,-2435
C08890=4308,28716,-32661,629,-26371,-2438
C08891=4315,28711,-32667,628,-26369,-2441
C08892=4322,28706,-32673,627,-26368,-2444
C08893=4327,28702,-32679,626,-26366,-2446
C08894=4318,28700,-32680,628,-26366,-2442
C08895=4311,28705,-32674,629,-26367,-2439
C08896=4303,28708,-32671,630,-26368,-2436
C08897=4294,28708,-32671,631,-26368,-2433
C08898=4287,28713,-32665,632,-26370,-2430
C08899=4279,28714,-32664,633,-26370,-2427
C08900=4270,28713,-32666,635,-26370,-2423
C08901=4261,28713,-32665,636,-26370,-2420
C08902=4254,28718,-32659,637,-26372,-2417
C08903=4246,28719,-32658,638,-26372,-2414
C08904=4237,28717,-32660,640,-26371,-2411
C08905=4227,28716,-32661,641,-26371,-2407
C08906=4219,28716,-32661,642,-26371,-2404
C08907=4212,28721,-32655,643,-26373,-2401
C08908=4203,28722,-32654,644,-26373,-2398
C08909=4194,28721,-32656,646,-26372,-2394
C08910=4185,28720,-32657,647,-26372,-2391
C08911=4176,28718,-32659,649,-26371,-2387
C08912=4167,28717,-32661,650,-26371,-2384
C08913=4158,28716,-32662,651,-26370,-2380
C08914=4149,28714,-32664,653,-26370,-2377
C08915=4140,28713,-32665,654,-26369,-2373
C08916=4130,28712,-32667,655,-26369,-2370
C08917=4121,28710,-32669,657,-26368,-2366
C08918=4113,28707,-32672,658,-26367,-2363
C08919=4107,28700,-32681,659,-26364,-2361
C08920=4099,28698,-32684,660,-26363,-2358
C08921=4090,28696,-32686,662,-26363,-2354
C08922=4084,28699,-31282,662,-26364,-2352
C08923=-41004,59868,4099,4900,-34257,16705
C08924=-41004,59868,1099,4900,-34257,16705
C08925=-41004,64596,1380,5213,-31659,16463
C08926=-41004,59868,1099,4900,-34257,16705
C08927=-41004,59868,9099,4900,-34257,16705
C08928=4084,28699,-28682,662,-26364,-2352
C08929=4084,28699,-32682,662,-26364,-2352
C08930=4084,28699,-31282,662,-26364,-2352
C08931=3915,29102,-28195,684,-26512,-2284
C08932=3915,29102,-32195,684,-26512,-2284
C08933=3904,29108,-32188,685,-26514,-2280
C08934=3892,29121,-32172,687,-26519,-2275
C08935=3881,29134,-32157,688,-26524,-2271
C08936=3866,29145,-32143,691,-26528,-2265
C08937=3848,29149,-32138,693,-26529,-2258
C08938=3831,29156,-32130,696,-26532,-2252
C08939=3811,29154,-32133,699,-26530,-2244
C08940=3791,29151,-32137,702,-26529,-2236
C08941=3771,29148,-32140,705,-26528,-2228
C08942=3752,29146,-32143,708,-26527,-2221
C08943=3736,29157,-32130,710,-26531,-2215
C08944=3718,29160,-32125,712,-26532,-2208
C08945=3701,29166,-32118,715,-26534,-2201
C08946=3681,29163,-32122,718,-26533,-2193
C08947=3665,29171,-32113,720,-26536,-2187
C08948=3644,29168,-32117,723,-26535,-2179
C08949=3627,29172,-32112,726,-26536,-2172
C08950=3613,29163,-32122,728,-26533,-2167
C08951=3593,29160,-32126,731,-26531,-2159
C08952=3578,29149,-32140,733,-26527,-2154
C08953=3564,29137,-32155,735,-26522,-2148
C08954=3551,29122,-32173,737,-26517,-2143
C08955=3538,29107,-32191,740,-26511,-2138
C08956=3526,29092,-32209,741,-26505,-2134
C08957=3527,29074,-32231,741,-26499,-2135
C08958=3519,29058,-32250,743,-26493,-2132
C08959=3525,29042,-32270,742,-26487,-2134
C08960=3521,29035,-32278,743,-26484,-2132
C08961=3500,29032,-32281,746,-26483,-2125
C08962=3499,29050,-32259,746,-26490,-2124
C08963=3497,29069,-32237,746,-26497,-2123
C08964=3506,29084,-32218,744,-26503,-2126
C08965=3506,29102,-32197,744,-26509,-2126
C08966=3513,29118,-32177,743,-26515,-2129
C08967=3522,29134,-32158,742,-26521,-2132
C08968=3530,29150,-32138,740,-26527,-2135
C08969=3543,29165,-32120,738,-26533,-2140
C08970=3559,29175,-32109,736,-26536,-2146
C08971=3574,29186,-32095,733,-26541,-2152
C08972=3594,29189,-32091,730,-26542,-2160
C08973=3614,29192,-32087,727,-26543,-2167
C08974=3634,29195,-32084,724,-26545,-2175
C08975=3654,29197,-32081,722,-26545,-2183
C08976=3670,29191,-32089,719,-26543,-2189
C08977=3691,29194,-32085,716,-26544,-2197
C08978=3707,29186,-32094,714,-26542,-2203
C08979=3725,29182,-32099,711,-26540,-2210
C08980=3744,29182,-32099,708,-26541,-2218
C08981=3761,29175,-32108,706,-26538,-2224
C08982=3781,29178,-32104,703,-26539,-2232
C08983=3801,29181,-32101,700,-26540,-2240
C08984=3819,29178,-32104,697,-26540,-2247
C08985=3837,29176,-32106,695,-26539,-2254
C08986=3854,29170,-32113,692,-26537,-2260
C08987=3872,29167,-32117,689,-26536,-2267
C08988=3888,29156,-32130,687,-26532,-2273
C08989=3903,29145,-32143,685,-26528,-2279
C08990=3912,29131,-32160,684,-26523,-2283
C08991=3921,29119,-32175,683,-26518,-2286
C08992=3915,29102,-32195,684,-26512,-2284
C08993=3915,29102,-30795,684,-26512,-2284
C08994=3764,29338,-27910,704,-26599,-2224
C08995=3764,29338,-31910,704,-26599,-2224
C08996=3743,29335,-31914,707,-26597,-2216
C08997=3721,29332,-31918,710,-26596,-2208
C08998=3700,29329,-31922,713,-26595,-2200
C08999=3684,29318,-31935,716,-26590,-2193
C09000=3663,29314,-31940,719,-26589,-2185
C09001=3641,29311,-31944,722,-26588,-2177
C09002=3623,29318,-31935,725,-26590,-2170
C09003=3602,29315,-31939,728,-26589,-2162
C09004=3581,29312,-31943,731,-26587,-2154
C09005=3561,29314,-31940,734,-26588,-2146
C09006=3542,29315,-31938,737,-26589,-2139
C09007=3520,29312,-31942,740,-26587,-2130
C09008=3499,29309,-31946,743,-26586,-2122
C09009=3478,29306,-31950,746,-26585,-2114
C09010=3456,29303,-31954,750,-26583,-2106
C09011=3442,29308,-31947,752,-26585,-2100
C09012=3449,29321,-31932,750,-26590,-2103
C09013=3471,29324,-31928,747,-26591,-2111
C09014=3488,29333,-31917,745,-26595,-2118
C09015=3506,29343,-31905,742,-26599,-2125
C09016=3524,29351,-31895,739,-26602,-2132
C09017=3545,29354,-31891,736,-26603,-2140
C09018=3565,29359,-31885,733,-26605,-2148
C09019=3583,29369,-31873,730,-26609,-2154
C09020=3604,29372,-31869,727,-26610,-2162
C09021=3621,29382,-31857,725,-26614,-2169
C09022=3641,29387,-31851,722,-26616,-2177
C09023=3663,29390,-31847,718,-26617,-2185
C09024=3684,29393,-31844,715,-26619,-2193
C09025=3705,29396,-31840,712,-26620,-2201
C09026=3727,29400,-31836,709,-26621,-2210
C09027=3748,29403,-31832,706,-26622,-2218
C09028=3769,29406,-31828,702,-26624,-2226
C09029=3790,29409,-31825,699,-26625,-2234
C09030=3812,29412,-31821,696,-26626,-2242
C09031=3830,29406,-31828,693,-26624,-2249
C09032=3851,29408,-31825,690,-26625,-2258
C09033=3872,29411,-31822,687,-26626,-2266
C09034=3891,29407,-31826,684,-26625,-2273
C09035=3912,29407,-31826,681,-26625,-2281
C09036=3930,29400,-31834,679,-26623,-2288
C09037=3951,29403,-31831,676,-26624,-2296
C09038=3972,29406,-31827,673,-26625,-2304
C09039=3994,29409,-31823,669,-26627,-2313
C09040=4011,29401,-31833,667,-26624,-2319
C09041=4004,29384,-31854,668,-26617,-2317
C09042=3983,29379,-31860,671,-26615,-2309
C09043=3962,29376,-31863,674,-26614,-2301
C09044=3944,29383,-31855,677,-26617,-2294
C09045=3923,29380,-31859,680,-26615,-2285
C09046=3901,29377,-31863,683,-26614,-2277
C09047=3880,29374,-31866,686,-26613,-2269
C09048=3862,29381,-31858,689,-26615,-2262
C09049=3842,29380,-31859,692,-26615,-2254
C09050=3823,29385,-31854,695,-26616,-2247
C09051=3806,29375,-31865,697,-26613,-2240
C09052=3810,29359,-31885,697,-26607,-2242
C09053=3801,29353,-31892,698,-26604,-2239
C09054=3782,29347,-31899,701,-26602,-2231
C09055=3764,29338,-31910,704,-26599,-2224
C09056=3764,29338,-30510,704,-26599,-2224
C09057=3751,29346,-27901,706,-26601,-2219
C09058=3751,29346,-31901,706,-26601,-2219
C09059=3756,29349,-31897,705,-26603,-2221
C09060=3760,29354,-31891,704,-26604,-2223
C09061=3764,29359,-31885,704,-26606,-2224
C09062=3769,29364,-31879,703,-26608,-2226
C09063=3772,29368,-31874,702,-26610,-2227
C09064=3767,29372,-31869,703,-26611,-2225
C09065=3762,29375,-31865,704,-26612,-2223
C09066=3757,29379,-31861,705,-26614,-2221
C09067=3751,29383,-31857,705,-26615,-2219
C09068=3745,29383,-31856,706,-26615,-2217
C09069=3739,29382,-31857,707,-26615,-2214
C09070=3732,29381,-31858,708,-26614,-2212
C09071=3726,29380,-31859,709,-26614,-2209
C09072=3719,29379,-31860,710,-26614,-2207
C09073=3713,29378,-31862,711,-26613,-2204
C09074=3706,29378,-31863,712,-26613,-2202
C09075=3700,29377,-31864,713,-26612,-2199
C09076=3693,29376,-31865,714,-26612,-2197
C09077=3687,29375,-31866,715,-26612,-2194
C09078=3680,29374,-31867,716,-26611,-2192
C09079=3674,29373,-31869,717,-26611,-2189
C09080=3667,29372,-31870,718,-26610,-2187
C09081=3660,29371,-31871,719,-26610,-2184
C09082=3654,29370,-31872,720,-26610,-2182
C09083=3647,29369,-31873,721,-26609,-2179
C09084=3641,29368,-31874,722,-26609,-2177
C09085=3635,29366,-31877,723,-26608,-2174
C09086=3631,29361,-31883,723,-26606,-2173
C09087=3626,29356,-31888,724,-26604,-2171
C09088=3620,29355,-31890,725,-26604,-2169
C09089=3613,29355,-31891,726,-26604,-2166
C09090=3607,29354,-31892,727,-26603,-2164
C09091=3602,29349,-31897,728,-26602,-2162
C09092=3598,29345,-31903,728,-26600,-2160
C09093=3597,29339,-31910,729,-26598,-2160
C09094=3597,29333,-31917,729,-26596,-2160
C09095=3602,29330,-31921,728,-26594,-2162
C09096=3607,29326,-31925,727,-26593,-2164
C09097=3613,29326,-31926,726,-26593,-2166
C09098=3620,29327,-30524,725,-26593,-2169
C09099=-41004,59868,4099,4900,-34257,16705
C09100=-41004,59868,1099,4900,-34257,16705
C09101=-41004,64596,1380,5213,-31659,16463
C09102=-41004,59868,1099,4900,-34257,16705
C09103=-41004,59868,9099,4900,-34257,16705
C09104=3620,29327,-27924,725,-26593,-2169
C09105=3620,29327,-31924,725,-26593,-2169
C09106=3627,29328,-31923,724,-26594,-2171
C09107=3633,29329,-31922,723,-26594,-2174
C09108=3640,29330,-31921,722,-26595,-2176
C09109=3646,29331,-31920,721,-26595,-2179
C09110=3653,29332,-31919,720,-26595,-2181
C09111=3659,29332,-31917,719,-26596,-2184
C09112=3666,29333,-31916,718,-26596,-2186
C09113=3672,29334,-31915,717,-26597,-2189
C09114=3679,29335,-31914,716,-26597,-2191
C09115=3685,29336,-31913,716,-26597,-2194
C09116=3692,29337,-31912,715,-26598,-2197
C09117=3699,29338,-31910,714,-26598,-2199
C09118=3705,29339,-31909,713,-26599,-2202
C09119=3712,29340,-31908,712,-26599,-2204
C09120=3718,29341,-31907,711,-26599,-2207
C09121=3725,29342,-31906,710,-26600,-2209
C09122=3731,29343,-31905,709,-26600,-2212
C09123=3738,29344,-31903,708,-26601,-2214
C09124=3744,29345,-31902,707,-26601,-2217
C09125=3751,29346,-31901,706,-26601,-2219
C09126=3751,29346,-30501,706,-26601,-2219
C09127=3711,29493,-27723,710,-26656,-2203
C09128=3711,29493,-31723,710,-26656,-2203
C09129=3703,29492,-31724,711,-26655,-2200
C09130=3694,29491,-31726,713,-26655,-2197
C09131=3686,29490,-31727,714,-26654,-2193
C09132=3680,29494,-31722,715,-26656,-2191
C09133=3673,29497,-31718,716,-26657,-2188
C09134=3664,29495,-31720,717,-26656,-2185
C09135=3659,29489,-31728,718,-26654,-2183
C09136=3653,29485,-31733,719,-26652,-2180
C09137=3644,29483,-31735,720,-26652,-2177
C09138=3636,29482,-31736,721,-26651,-2174
C09139=3627,29481,-31738,723,-26651,-2171
C09140=3619,29480,-31739,724,-26650,-2167
C09141=3611,29478,-31741,725,-26650,-2164
C09142=3603,29476,-31743,726,-26649,-2161
C09143=3597,29470,-31751,727,-26646,-2159
C09144=3591,29466,-31756,728,-26645,-2157
C09145=3583,29464,-31759,729,-26644,-2154
C09146=3578,29458,-31766,730,-26642,-2152
C09147=3571,29454,-31771,731,-26640,-2149
C09148=3562,29452,-31773,733,-26640,-2146
C09149=3554,29451,-31774,734,-26639,-2142
C09150=3553,29459,-31765,734,-26642,-2142
C09151=3557,29465,-31757,733,-26644,-2144
C09152=3563,29472,-31749,732,-26647,-2146
C09153=3568,29478,-31742,731,-26649,-2148
C09154=3574,29483,-31736,730,-26651,-2150
C09155=3582,29484,-31734,729,-26652,-2153
C09156=3588,29491,-31726,728,-26654,-2155
C09157=3594,29495,-31721,727,-26656,-2158
C09158=3603,29496,-31719,726,-26656,-2161
C09159=3611,29498,-31718,725,-26657,-2164
C09160=3619,29499,-31716,724,-26657,-2167
C09161=3628,29500,-31715,722,-26658,-2171
C09162=3636,29501,-31713,721,-26658,-2174
C09163=3645,29503,-31712,720,-26659,-2177
C09164=3653,29504,-31710,719,-26659,-2180
C09165=3661,29505,-31709,717,-26660,-2184
C09166=3670,29506,-31707,716,-26660,-2187
C09167=3678,29507,-31706,715,-26661,-2190
C09168=3687,29509,-31704,714,-26661,-2193
C09169=3695,29510,-31703,712,-26662,-2197
C09170=3703,29511,-31701,711,-26662,-2200
C09171=3712,29512,-31700,710,-26663,-2203
C09172=3720,29513,-31698,709,-26663,-2206
C09173=3728,29515,-31697,707,-26664,-2210
C09174=3737,29516,-31695,706,-26664,-2213
C09175=3745,29517,-31694,705,-26665,-2216
C09176=3754,29518,-31692,704,-26665,-2219
C09177=3761,29516,-31695,703,-26665,-2222
C09178=3767,29511,-31701,702,-26663,-2225
C09179=3774,29507,-31706,701,-26661,-2227
C09180=3778,29503,-31711,700,-26660,-2229
C09181=3770,29501,-31712,701,-26659,-2226
C09182=3762,29500,-31714,703,-26659,-2222
C09183=3753,29499,-31715,704,-26658,-2219
C09184=3745,29498,-31717,705,-26658,-2216
C09185=3736,29497,-31718,706,-26657,-2213
C09186=3728,29495,-31720,708,-26657,-2209
C09187=3720,29494,-31721,709,-26656,-2206
C09188=3711,29493,-31723,710,-26656,-2203
C09189=3711,29493,-30323,710,-26656,-2203
C09190=4824,28052,-29464,558,-26127,-2641
C09191=4824,28052,-33464,558,-26127,-2641
C09192=4855,28055,-33460,553,-26129,-2653
C09193=4840,28038,-33481,555,-26122,-2647
C09194=4818,28012,-33512,559,-26113,-2639
C09195=4792,27993,-33535,563,-26106,-2629
C09196=4770,27968,-33565,566,-26096,-2621
C09197=4745,27948,-33589,570,-26089,-2611
C09198=4722,27924,-33619,574,-26079,-2602
C09199=4700,27899,-33650,578,-26070,-2594
C09200=4678,27873,-33680,581,-26060,-2586
C09201=4652,27854,-33703,585,-26053,-2576
C09202=4630,27829,-33734,589,-26044,-2568
C09203=4608,27804,-33765,592,-26034,-2559
C09204=4584,27782,-33791,596,-26026,-2550
C09205=4560,27760,-33818,600,-26017,-2541
C09206=4535,27741,-33841,604,-26010,-2531
C09207=4509,27722,-33864,608,-26003,-2521
C09208=4484,27701,-33890,612,-25995,-2512
C09209=4460,27678,-33917,615,-25986,-2503
C09210=4431,27664,-33934,620,-25981,-2492
C09211=4405,27645,-33957,624,-25974,-2482
C09212=4378,27628,-33978,628,-25967,-2472
C09213=4348,27614,-33995,633,-25962,-2460
C09214=4319,27601,-34011,637,-25957,-2449
C09215=4289,27588,-34027,642,-25952,-2438
C09216=4256,27581,-34035,647,-25949,-2425
C09217=4226,27568,-34051,652,-25944,-2414
C09218=4197,27554,-34068,656,-25939,-2402
C09219=4162,27549,-34074,661,-25937,-2389
C09220=4133,27535,-34090,666,-25932,-2378
C09221=4103,27522,-34107,670,-25927,-2367
C09222=4069,27517,-34113,676,-25925,-2353
C09223=4092,27530,-34097,672,-25929,-2362
C09224=4121,27543,-34081,668,-25935,-2373
C09225=4150,27557,-34064,663,-25940,-2385
C09226=4184,27563,-34056,658,-25942,-2398
C09227=4214,27576,-34041,653,-25947,-2409
C09228=4244,27590,-34025,649,-25953,-2420
C09229=4273,27603,-34008,644,-25958,-2431
C09230=4304,27615,-33994,640,-25962,-2443
C09231=4333,27628,-33978,635,-25967,-2455
C09232=4363,27640,-33963,630,-25972,-2466
C09233=4390,27658,-33941,626,-25979,-2476
C09234=4419,27672,-33924,622,-25984,-2487
C09235=4445,27691,-33901,618,-25991,-2497
C09236=4471,27710,-33878,614,-25999,-2507
C09237=4497,27729,-33855,610,-26006,-2517
C09238=4523,27748,-33832,605,-26013,-2527
C09239=4545,27774,-33801,602,-26023,-2535
C09240=4571,27793,-33778,598,-26030,-2545
C09241=4593,27818,-33748,594,-26039,-2553
C09242=4615,27843,-33717,591,-26049,-2562
C09243=4637,27869,-33686,587,-26058,-2570
C09244=4663,27888,-33663,583,-26065,-2580
C09245=4685,27913,-33633,580,-26075,-2588
C09246=4707,27938,-33602,576,-26084,-2596
C09247=4733,27957,-33579,572,-26092,-2606
C09248=4755,27982,-33548,569,-26101,-2615
C09249=4777,28008,-33518,565,-26111,-2623
C09250=4802,28027,-33495,561,-26118,-2633
C09251=4824,28052,-33464,558,-26127,-2641
C09252=4824,28052,-32064,558,-26127,-2641
C09253=4904,27866,-29689,547,-26059,-2673
C09254=4904,27866,-33689,547,-26059,-2673
C09255=4888,27838,-33723,550,-26048,-2667
C09256=4873,27810,-33757,552,-26038,-2661
C09257=4858,27782,-33791,555,-26027,-2655
C09258=4835,27755,-33823,559,-26017,-2647
C09259=4812,27729,-33856,562,-26007,-2638
C09260=4789,27702,-33888,566,-25997,-2629
C09261=4765,27676,-33920,570,-25987,-2620
C09262=4738,27655,-33944,574,-25980,-2610
C09263=4711,27635,-33969,578,-25972,-2600
C09264=4685,27615,-33994,582,-25964,-2590
C09265=4657,27594,-34018,587,-25956,-2579
C09266=4628,27578,-34038,591,-25950,-2568
C09267=4599,27560,-34060,596,-25943,-2557
C09268=4572,27541,-34083,600,-25936,-2547
C09269=4541,27527,-34100,605,-25931,-2535
C09270=4510,27513,-34117,610,-25925,-2523
C09271=4479,27499,-34134,614,-25920,-2511
C09272=4448,27485,-34151,619,-25915,-2499
C09273=4417,27471,-34168,624,-25909,-2488
C09274=4383,27462,-32779,629,-25906,-2475
C09275=-41004,59868,4099,4900,-34257,16705
C09276=-41004,59868,1099,4900,-34257,16705
C09277=-41004,64596,1380,5213,-31659,16463
C09278=-41004,59868,1099,4900,-34257,16705
C09279=-41004,59868,9099,4900,-34257,16705
C09280=4383,27462,-30179,629,-25906,-2475
C09281=4383,27462,-34179,629,-25906,-2475
C09282=4352,27448,-34196,634,-25900,-2463
C09283=4318,27438,-34208,639,-25896,-2450
C09284=4287,27424,-34225,644,-25891,-2438
C09285=4255,27412,-34240,649,-25886,-2426
C09286=4220,27404,-34250,654,-25883,-2412
C09287=4188,27390,-34266,659,-25878,-2400
C09288=4157,27376,-34283,664,-25873,-2388
C09289=4121,27371,-34289,669,-25871,-2374
C09290=4090,27357,-34306,674,-25865,-2363
C09291=4053,27352,-34312,680,-25863,-2349
C09292=4076,27368,-34293,676,-25869,-2357
C09293=4109,27379,-34280,671,-25874,-2370
C09294=4140,27393,-34263,666,-25879,-2382
C09295=4177,27398,-34256,661,-25881,-2396
C09296=4208,27412,-34239,656,-25886,-2408
C09297=4239,27426,-34223,651,-25892,-2420
C09298=4274,27433,-34213,646,-25895,-2433
C09299=4306,27446,-34199,641,-25899,-2445
C09300=4337,27460,-34182,636,-25905,-2457
C09301=4368,27474,-34165,631,-25910,-2469
C09302=4402,27484,-34153,626,-25914,-2482
C09303=4433,27498,-34136,621,-25919,-2494
C09304=4464,27512,-34118,616,-25925,-2505
C09305=4495,27526,-34101,612,-25930,-2517
C09306=4526,27540,-34084,607,-25936,-2529
C09307=4557,27554,-34067,602,-25941,-2541
C09308=4585,27572,-34046,598,-25948,-2552
C09309=4616,27586,-34029,593,-25953,-2564
C09310=4646,27602,-34009,588,-25959,-2575
C09311=4673,27623,-33984,584,-25967,-2585
C09312=4700,27643,-33959,580,-25975,-2595
C09313=4727,27663,-33935,576,-25982,-2606
C09314=4750,27690,-33903,572,-25992,-2614
C09315=4777,27710,-33878,568,-26000,-2625
C09316=4800,27736,-33846,564,-26010,-2633
C09317=4823,27763,-33814,560,-26020,-2642
C09318=4846,27789,-33782,557,-26030,-2651
C09319=4862,27818,-33748,554,-26040,-2657
C09320=4877,27846,-33714,552,-26051,-2662
C09321=4904,27866,-33689,547,-26059,-2673
C09322=4904,27866,-32289,547,-26059,-2673
C09323=3787,27402,-30253,719,-25880,-2246
C09324=3787,27402,-34253,719,-25880,-2246
C09325=3775,27398,-34257,721,-25879,-2241
C09326=3757,27396,-34260,724,-25878,-2234
C09327=3743,27403,-34251,726,-25881,-2229
C09328=3728,27407,-34247,728,-25882,-2223
C09329=3715,27416,-34236,730,-25885,-2218
C09330=3699,27418,-34233,732,-25886,-2212
C09331=3684,27423,-34227,734,-25888,-2206
C09332=3667,27421,-34230,737,-25887,-2199
C09333=3651,27424,-34226,739,-25888,-2193
C09334=3635,27426,-34224,742,-25889,-2187
C09335=3619,27428,-34221,744,-25889,-2181
C09336=3604,27431,-34217,746,-25890,-2175
C09337=3588,27432,-34216,749,-25891,-2169
C09338=3573,27436,-34211,751,-25892,-2163
C09339=3559,27443,-34203,753,-25895,-2158
C09340=3543,27445,-34200,755,-25895,-2152
C09341=3527,27449,-34196,758,-25896,-2146
C09342=3514,27457,-34187,760,-25899,-2140
C09343=3500,27464,-34178,762,-25902,-2135
C09344=3484,27468,-34173,764,-25903,-2129
C09345=3471,27477,-34162,766,-25907,-2124
C09346=3455,27479,-34160,768,-25907,-2118
C09347=3442,27488,-34149,770,-25911,-2113
C09348=3429,27497,-34138,772,-25914,-2107
C09349=3413,27499,-34135,774,-25915,-2101
C09350=3399,27509,-34124,776,-25918,-2096
C09351=3386,27518,-34113,778,-25921,-2091
C09352=3373,27527,-34102,780,-25925,-2086
C09353=3366,27540,-34087,781,-25929,-2083
C09354=3355,27550,-34075,783,-25933,-2079
C09355=3360,27553,-34070,782,-25934,-2081
C09356=3373,27544,-34081,780,-25931,-2086
C09357=3387,27535,-34092,778,-25928,-2091
C09358=3400,27526,-34103,776,-25924,-2096
C09359=3414,27518,-34112,774,-25922,-2102
C09360=3429,27515,-34117,772,-25920,-2107
C09361=3442,27505,-34128,770,-25917,-2113
C09362=3458,27503,-34130,767,-25916,-2119
C09363=3472,27494,-34141,766,-25913,-2124
C09364=3485,27485,-34152,764,-25910,-2129
C09365=3501,27483,-34155,761,-25909,-2135
C09366=3515,27476,-34164,759,-25906,-2141
C09367=3530,27472,-34168,757,-25905,-2147
C09368=3543,27463,-34179,755,-25902,-2152
C09369=3559,27461,-34182,753,-25901,-2158
C09370=3572,27452,-34193,751,-25898,-2163
C09371=3588,27448,-34197,749,-25896,-2169
C09372=3604,27447,-34198,746,-25896,-2175
C09373=3619,27443,-34203,744,-25895,-2181
C09374=3636,27445,-34200,741,-25896,-2188
C09375=3652,27441,-34205,739,-25894,-2194
C09376=3668,27440,-34206,737,-25894,-2200
C09377=3683,27437,-34210,734,-25893,-2206
C09378=3699,27435,-34212,732,-25892,-2212
C09379=3713,27427,-34222,730,-25890,-2217
C09380=3728,27424,-34226,728,-25888,-2223
C09381=3744,27422,-34228,725,-25888,-2229
C09382=3758,27415,-34237,723,-25885,-2235
C09383=3773,27411,-34242,721,-25884,-2241
C09384=3787,27402,-34253,719,-25880,-2246
C09385=3787,27402,-32853,719,-25880,-2246
C09386=6040,32559,-23996,349,-27818,-3091
C09387=6040,32559,-27996,349,-27818,-3091
C09388=6037,32580,-27971,349,-27826,-3089
C09389=6034,32600,-27946,349,-27834,-3088
C09390=6031,32621,-27921,350,-27841,-3087
C09391=6024,32638,-27900,351,-27848,-3084
C09392=6016,32656,-27878,351,-27854,-3081
C09393=6013,32677,-27853,352,-27862,-3080
C09394=6001,32692,-27835,353,-27868,-3075
C09395=5998,32712,-27810,354,-27875,-3074
C09396=5986,32727,-27792,355,-27881,-3069
C09397=5983,32748,-27767,356,-27888,-3068
C09398=5971,32763,-27749,357,-27894,-3063
C09399=5968,32783,-27724,358,-27901,-3062
C09400=5956,32798,-27706,359,-27907,-3057
C09401=5950,32817,-27683,360,-27914,-3055
C09402=5941,32834,-27663,361,-27920,-3051
C09403=5935,32853,-27640,362,-27927,-3049
C09404=5926,32869,-27620,363,-27933,-3045
C09405=5921,32889,-27597,364,-27940,-3043
C09406=5910,32905,-27577,365,-27946,-3039
C09407=5898,32920,-27559,367,-27952,-3034
C09408=5889,32937,-27538,368,-27958,-3031
C09409=5883,32956,-27516,369,-27965,-3028
C09410=5871,32971,-27497,371,-27971,-3024
C09411=5864,32989,-27476,372,-27977,-3021
C09412=5853,33005,-27456,373,-27983,-3016
C09413=5844,33021,-27436,374,-27989,-3013
C09414=5832,33037,-27418,376,-27995,-3008
C09415=5821,33053,-27398,377,-28001,-3004
C09416=5817,33072,-27375,378,-28008,-3002
C09417=5824,33076,-27370,377,-28010,-3005
C09418=5838,33062,-27387,375,-28004,-3011
C09419=5851,33047,-27405,373,-27999,-3015
C09420=5856,33028,-27428,373,-27992,-3018
C09421=5867,33012,-27448,371,-27986,-3022
C09422=5878,32996,-27467,370,-27980,-3026
C09423=5888,32980,-27486,368,-27974,-3030
C09424=5893,32960,-27510,368,-27967,-3032
C09425=5905,32945,-27528,366,-27961,-3037
C09426=5917,32930,-27546,364,-27956,-3042
C09427=5924,32912,-27568,363,-27949,-3044
C09428=5932,32895,-27589,362,-27943,-3048
C09429=5939,32876,-27612,362,-27936,-3050
C09430=5947,32859,-27632,360,-27930,-3054
C09431=5960,32844,-27651,359,-27924,-3058
C09432=5962,32823,-27675,358,-27916,-3060
C09433=5975,32808,-27694,357,-27911,-3064
C09434=5979,32789,-27718,356,-27904,-3066
C09435=5990,32773,-27737,355,-27898,-3070
C09436=5993,32753,-27761,354,-27890,-3072
C09437=6005,32737,-27780,353,-27885,-3076
C09438=6008,32717,-27804,352,-27877,-3078
C09439=6020,32702,-27823,351,-27871,-3082
C09440=6023,32681,-27848,350,-27864,-3084
C09441=6033,32665,-27867,349,-27858,-3088
C09442=6038,32646,-27891,348,-27851,-3090
C09443=6041,32625,-27915,348,-27843,-3091
C09444=6052,32610,-27934,347,-27837,-3095
C09445=6048,32592,-27956,347,-27830,-3094
C09446=6048,32572,-27980,347,-27823,-3094
C09447=6040,32559,-26596,349,-27818,-3091
C09448=-41004,59868,4099,4900,-34257,16705
C09449=-41004,59868,1099,4900,-34257,16705
C09450=-41004,64596,1380,5213,-31659,16463
C09451=-41004,59868,1099,4900,-34257,16705
C09452=-41004,59868,9099,4900,-34257,16705
C09453=6040,32559,-23996,349,-27818,-3091
C09454=6040,32559,-27996,349,-27818,-3091
C09455=6040,32559,-26596,349,-27818,-3091
C09456=6356,32692,-23833,302,-27871,-3213
C09457=6356,32692,-27833,302,-27871,-3213
C09458=6363,32712,-27808,301,-27879,-3216
C09459=6363,32734,-27781,301,-27887,-3216
C09460=6370,32754,-27757,300,-27895,-3218
C09461=6377,32775,-27732,299,-27902,-3221
C09462=6385,32795,-27707,298,-27910,-3224
C09463=6392,32815,-27682,297,-27918,-3227
C09464=6399,32836,-27658,296,-27925,-3230
C09465=6406,32856,-27633,294,-27933,-3232
C09466=6414,32876,-27608,293,-27941,-3235
C09467=6417,32898,-27582,293,-27949,-3236
C09468=6424,32918,-27557,292,-27957,-3239
C09469=6431,32938,-27533,291,-27964,-3242
C09470=6428,32961,-27505,291,-27973,-3240
C09471=6424,32984,-27477,291,-27981,-3239
C09472=6431,33004,-27453,290,-27989,-3242
C09473=6428,33027,-27425,291,-27997,-3240
C09474=6416,33045,-27404,292,-28004,-3235
C09475=6412,33067,-27376,293,-28012,-3234
C09476=6409,33090,-27348,293,-28021,-3232
C09477=6416,33111,-27324,292,-28029,-3235
C09478=6412,33133,-27296,292,-28037,-3234
C09479=6409,33156,-27268,293,-28046,-3232
C09480=6406,33179,-27241,293,-28054,-3231
C09481=6402,33202,-27213,294,-28063,-3230
C09482=6399,33225,-27185,294,-28071,-3228
C09483=6406,33245,-27161,293,-28079,-3231
C09484=6403,33268,-27133,293,-28087,-3230
C09485=6399,33291,-27105,294,-28096,-3228
C09486=6398,33313,-27078,294,-28104,-3228
C09487=6406,33329,-27058,293,-28111,-3231
C09488=6416,33311,-27081,291,-28104,-3235
C09489=6420,33288,-27108,291,-28095,-3236
C09490=6414,33267,-27134,292,-28087,-3234
C09491=6416,33245,-27161,291,-28079,-3235
C09492=6419,33222,-27188,291,-28070,-3236
C09493=6423,33199,-27216,291,-28062,-3238
C09494=6426,33176,-27244,290,-28053,-3239
C09495=6429,33154,-27271,290,-28045,-3240
C09496=6422,33133,-27296,291,-28037,-3238
C09497=6426,33110,-27324,291,-28029,-3239
C09498=6429,33088,-27352,290,-28020,-3240
C09499=6432,33065,-27379,290,-28012,-3242
C09500=6436,33042,-27407,289,-28003,-3243
C09501=6439,33019,-27435,289,-27995,-3245
C09502=6443,32996,-27462,289,-27986,-3246
C09503=6446,32974,-27490,288,-27978,-3247
